DATA_BLOCK "PackMLCfg"   // DB31603
TITLE = CPG_PackMLCfg
{ S7_Optimized_Access := 'TRUE' }
AUTHOR : tech.team.motioncontrol@siemens.com
FAMILY : CPG
VERSION : 1.0
// Support: tech.team.motioncontrol@siemens.com
// Fax: +49 (0) 9131/98-1297
// stored: AutoNumber true, DBAccessibleFromOPCUA true, DBAccessibleFromWebserver true, IsOnlyStoredInLoadMemory false, IsRetainMemResEnabled false, IsWriteProtectedInAS false, MemoryReserve 0
   VAR
      Cfg { S7_SetPoint := 'True'} : "typeLPMLV30_Configuration";   // PackML Configuration Data
      Names { S7_SetPoint := 'True'} : "typeLPMLV30_NamesConfiguration";   // PackML Names Data
      disable : Struct   // Bits used to disable TR88 UN & EMs
         UN : Bool;   // UN (1 = disable, 0= enable)
         EM00 : Struct   // EM00 (1 = disable, 0 = enable)
            EM : Bool;   // EMxx (1 = disable, 0 = enable)
            CM01 : Bool;   // CMxx (1 = disable, 0 = enable)
            CM02 : Bool;   // CMxx (1 = disable, 0 = enable)
            CM03 : Bool;   // CMxx (1 = disable, 0 = enable)
            CM04 : Bool;   // CMxx (1 = disable, 0 = enable)
            CM05 : Bool;   // CMxx (1 = disable, 0 = enable)
            CM06 : Bool;   // CMxx (1 = disable, 0 = enable)
            CM07 : Bool;   // CMxx (1 = disable, 0 = enable)
            CM08 : Bool;   // CMxx (1 = disable, 0 = enable)
            CM09 : Bool;   // CMxx (1 = disable, 0 = enable)
            CM10 : Bool;   // CMxx (1 = disable, 0 = enable)
         END_STRUCT;
         EM01 : Struct   // EM01 (1 = disable, 0 = enable)
            EM : Bool;   // EMxx (1 = disable, 0 = enable)
            CM01 : Bool;   // CMxx (1 = disable, 0 = enable)
            CM02 : Bool;   // CMxx (1 = disable, 0 = enable)
            CM03 : Bool;   // CMxx (1 = disable, 0 = enable)
            CM04 : Bool;   // CMxx (1 = disable, 0 = enable)
            CM05 : Bool;   // CMxx (1 = disable, 0 = enable)
            CM06 : Bool;   // CMxx (1 = disable, 0 = enable)
            CM07 : Bool;   // CMxx (1 = disable, 0 = enable)
            CM08 : Bool;   // CMxx (1 = disable, 0 = enable)
            CM09 : Bool;   // CMxx (1 = disable, 0 = enable)
            CM10 : Bool;   // CMxx (1 = disable, 0 = enable)
         END_STRUCT;
         EM02 : Struct   // EM02 (1 = disable, 0 = enable)
            EM : Bool;   // EMxx (1 = disable, 0 = enable)
            CM01 : Bool;   // CMxx (1 = disable, 0 = enable)
            CM02 : Bool;   // CMxx (1 = disable, 0 = enable)
            CM03 : Bool;   // CMxx (1 = disable, 0 = enable)
            CM04 : Bool;   // CMxx (1 = disable, 0 = enable)
            CM05 : Bool;   // CMxx (1 = disable, 0 = enable)
            CM06 : Bool;   // CMxx (1 = disable, 0 = enable)
            CM07 : Bool;   // CMxx (1 = disable, 0 = enable)
            CM08 : Bool;   // CMxx (1 = disable, 0 = enable)
            CM09 : Bool;   // CMxx (1 = disable, 0 = enable)
            CM10 : Bool;   // CMxx (1 = disable, 0 = enable)
         END_STRUCT;
         EM03 : Struct   // EM03 (1 = disable, 0 = enable)
            EM : Bool;   // EMxx (1 = disable, 0 = enable)
            CM01 : Bool;   // CMxx (1 = disable, 0 = enable)
            CM02 : Bool;   // CMxx (1 = disable, 0 = enable)
            CM03 : Bool;   // CMxx (1 = disable, 0 = enable)
            CM04 : Bool;   // CMxx (1 = disable, 0 = enable)
            CM05 : Bool;   // CMxx (1 = disable, 0 = enable)
            CM06 : Bool;   // CMxx (1 = disable, 0 = enable)
            CM07 : Bool;   // CMxx (1 = disable, 0 = enable)
            CM08 : Bool;   // CMxx (1 = disable, 0 = enable)
            CM09 : Bool;   // CMxx (1 = disable, 0 = enable)
            CM10 : Bool;   // CMxx (1 = disable, 0 = enable)
         END_STRUCT;
         EM04 : Struct   // EM04 (1 = disable, 0 = enable)
            EM : Bool;   // EMxx (1 = disable, 0 = enable)
            CM01 : Bool;   // CMxx (1 = disable, 0 = enable)
            CM02 : Bool;   // CMxx (1 = disable, 0 = enable)
            CM03 : Bool;   // CMxx (1 = disable, 0 = enable)
            CM04 : Bool;   // CMxx (1 = disable, 0 = enable)
            CM05 : Bool;   // CMxx (1 = disable, 0 = enable)
            CM06 : Bool;   // CMxx (1 = disable, 0 = enable)
            CM07 : Bool;   // CMxx (1 = disable, 0 = enable)
            CM08 : Bool;   // CMxx (1 = disable, 0 = enable)
            CM09 : Bool;   // CMxx (1 = disable, 0 = enable)
            CM10 : Bool;   // CMxx (1 = disable, 0 = enable)
         END_STRUCT;
         EM05 : Struct   // EM05 (1 = disable, 0 = enable)
            EM : Bool;   // EMxx (1 = disable, 0 = enable)
            CM01 : Bool;   // CMxx (1 = disable, 0 = enable)
            CM02 : Bool;   // CMxx (1 = disable, 0 = enable)
            CM03 : Bool;   // CMxx (1 = disable, 0 = enable)
            CM04 : Bool;   // CMxx (1 = disable, 0 = enable)
            CM05 : Bool;   // CMxx (1 = disable, 0 = enable)
            CM06 : Bool;   // CMxx (1 = disable, 0 = enable)
            CM07 : Bool;   // CMxx (1 = disable, 0 = enable)
            CM08 : Bool;   // CMxx (1 = disable, 0 = enable)
            CM09 : Bool;   // CMxx (1 = disable, 0 = enable)
            CM10 : Bool;   // CMxx (1 = disable, 0 = enable)
         END_STRUCT;
         EM06 : Struct   // EM06 (1 = disable, 0 = enable)
            EM : Bool;   // EMxx (1 = disable, 0 = enable)
            CM01 : Bool;   // CMxx (1 = disable, 0 = enable)
            CM02 : Bool;   // CMxx (1 = disable, 0 = enable)
            CM03 : Bool;   // CMxx (1 = disable, 0 = enable)
            CM04 : Bool;   // CMxx (1 = disable, 0 = enable)
            CM05 : Bool;   // CMxx (1 = disable, 0 = enable)
            CM06 : Bool;   // CMxx (1 = disable, 0 = enable)
            CM07 : Bool;   // CMxx (1 = disable, 0 = enable)
            CM08 : Bool;   // CMxx (1 = disable, 0 = enable)
            CM09 : Bool;   // CMxx (1 = disable, 0 = enable)
            CM10 : Bool;   // CMxx (1 = disable, 0 = enable)
         END_STRUCT;
         EM07 : Struct   // EM07 (1 = disable, 0 = enable)
            EM : Bool;   // EMxx (1 = disable, 0 = enable)
            CM01 : Bool;   // CMxx (1 = disable, 0 = enable)
            CM02 : Bool;   // CMxx (1 = disable, 0 = enable)
            CM03 : Bool;   // CMxx (1 = disable, 0 = enable)
            CM04 : Bool;   // CMxx (1 = disable, 0 = enable)
            CM05 : Bool;   // CMxx (1 = disable, 0 = enable)
            CM06 : Bool;   // CMxx (1 = disable, 0 = enable)
            CM07 : Bool;   // CMxx (1 = disable, 0 = enable)
            CM08 : Bool;   // CMxx (1 = disable, 0 = enable)
            CM09 : Bool;   // CMxx (1 = disable, 0 = enable)
            CM10 : Bool;   // CMxx (1 = disable, 0 = enable)
         END_STRUCT;
         EM08 : Struct   // EM08 (1 = disable, 0 = enable)
            EM : Bool;   // EMxx (1 = disable, 0 = enable)
            CM01 : Bool;   // CMxx (1 = disable, 0 = enable)
            CM02 : Bool;   // CMxx (1 = disable, 0 = enable)
            CM03 : Bool;   // CMxx (1 = disable, 0 = enable)
            CM04 : Bool;   // CMxx (1 = disable, 0 = enable)
            CM05 : Bool;   // CMxx (1 = disable, 0 = enable)
            CM06 : Bool;   // CMxx (1 = disable, 0 = enable)
            CM07 : Bool;   // CMxx (1 = disable, 0 = enable)
            CM08 : Bool;   // CMxx (1 = disable, 0 = enable)
            CM09 : Bool;   // CMxx (1 = disable, 0 = enable)
            CM10 : Bool;   // CMxx (1 = disable, 0 = enable)
         END_STRUCT;
         EM09 : Struct   // EM09 (1 = disable, 0 = enable)
            EM : Bool;   // EMxx (1 = disable, 0 = enable)
            CM01 : Bool;   // CMxx (1 = disable, 0 = enable)
            CM02 : Bool;   // CMxx (1 = disable, 0 = enable)
            CM03 : Bool;   // CMxx (1 = disable, 0 = enable)
            CM04 : Bool;   // CMxx (1 = disable, 0 = enable)
            CM05 : Bool;   // CMxx (1 = disable, 0 = enable)
            CM06 : Bool;   // CMxx (1 = disable, 0 = enable)
            CM07 : Bool;   // CMxx (1 = disable, 0 = enable)
            CM08 : Bool;   // CMxx (1 = disable, 0 = enable)
            CM09 : Bool;   // CMxx (1 = disable, 0 = enable)
            CM10 : Bool;   // CMxx (1 = disable, 0 = enable)
         END_STRUCT;
      END_STRUCT;
   END_VAR
BEGIN
   Names.unitModesNames[2,0] := 'Invalid';
   Names.unitModesNames[2,1] := 'Production';
   Names.unitModesNames[2,2] := 'Maintenance';
   Names.unitModesNames[2,3] := 'Manual';
   Names.unitModesNames[2,4] := 'User Mode 01';
   Names.statesNames[1,1] := 'Clearing';
   Names.statesNames[1,2] := 'Stopped';
   Names.statesNames[1,3] := 'Starting';
   Names.statesNames[1,4] := 'Idle';
   Names.statesNames[1,5] := 'Suspended';
   Names.statesNames[1,6] := 'Execute';
   Names.statesNames[1,7] := 'Stopping';
   Names.statesNames[1,8] := 'Aborting';
   Names.statesNames[1,9] := 'Aborted';
   Names.statesNames[1,10] := 'Holding';
   Names.statesNames[1,11] := 'Held';
   Names.statesNames[1,12] := 'UnHolding';
   Names.statesNames[1,13] := 'Suspending';
   Names.statesNames[1,14] := 'UnSuspending';
   Names.statesNames[1,15] := 'Resetting';
   Names.statesNames[1,16] := 'Completing';
   Names.statesNames[1,17] := 'Complete';
   Names.statesNames[2,0] := 'Undefined';
   Names.statesNames[2,1] := 'Limpiar';
   Names.statesNames[2,2] := 'Detenido';
   Names.statesNames[2,3] := 'Empezando';
   Names.statesNames[2,4] := 'Parado';
   Names.statesNames[2,5] := 'Interrumpido';
   Names.statesNames[2,6] := 'Correr';
   Names.statesNames[2,7] := 'Detener';
   Names.statesNames[2,8] := 'Anulando';
   Names.statesNames[2,9] := 'Anulado';
   Names.statesNames[2,10] := 'Mantener';
   Names.statesNames[2,11] := 'Mantenido';
   Names.statesNames[2,12] := 'Desmentener';
   Names.statesNames[2,13] := 'Interrumpir';
   Names.statesNames[2,14] := 'Desinterrumpir';
   Names.statesNames[2,15] := 'Reajustar';
   Names.statesNames[2,16] := 'Terminar';
   Names.statesNames[2,17] := 'Terminado';
END_DATA_BLOCK

DATA_BLOCK "RecipeCfg"   // DB1605
TITLE = CPG_RecipeCfg
{ S7_Optimized_Access := 'TRUE' }
AUTHOR : tech.team.motioncontrol@siemens.com
FAMILY : CPG
VERSION : 1.1
// Support: tech.team.motioncontrol@siemens.com
// stored: AutoNumber true, DBAccessibleFromOPCUA true, DBAccessibleFromWebserver true, IsOnlyStoredInLoadMemory false, IsRetainMemResEnabled false, IsWriteProtectedInAS false, MemoryReserve 0
   VAR
      setpoints_REAL { S7_SetPoint := 'True'} : Array[0.."CPG_NO_OF_SETPOINT_REAL_UPPER_LIM"] of "CPG_typeRecipeSetpoint_REAL";   // Array of setpoints of REAL
      setpoints_DINT { S7_SetPoint := 'True'} : Array[0.."CPG_NO_OF_SETPOINT_DINT_UPPER_LIM"] of "CPG_typeRecipeSetpoint_DINT";   // Array of setpoints of DINT
      setpoints_BOOL { S7_SetPoint := 'True'} : Array[0.."CPG_NO_OF_SETPOINT_BOOL_UPPER_LIM"] of "CPG_typeRecipeSetpoint_BOOL";   // Array of setpoints of BOOL
      setpoints_STRING { S7_SetPoint := 'True'} : Array[0.."CPG_NO_OF_SETPOINT_STRING_UPPER_LIM"] of "CPG_typeRecipeSetpoint_STRING";   // Array of setpoints of STRING
      recipeControl { S7_SetPoint := 'True'} : "CPG_typeRecipeControl";   // FB_Recipe_Control communicates to the setpoints via this tag
      recipeNames : Array[0.."CPG_NO_OF_RECIPE_UPPER_LIM"] of String[60];   // Array holding the names of all recipes
      recipeCumTimes : Array[0.."CPG_NO_OF_RECIPE_UPPER_LIM"] of Time;   // Array holding the cumulative time all recipes have been active
      recipeLastSaveTimes : Array[0.."CPG_NO_OF_RECIPE_UPPER_LIM"] of DTL;   // Array holding the last time each recipe was saved
   END_VAR
BEGIN
   setpoints_REAL[0].SetpointName[0] := 'LH 1 Length';
   setpoints_DINT[0].SetpointName[0] := 'DINT SP 0';
   setpoints_BOOL[0].SetpointName[0] := 'BOOL SP 0';
   setpoints_BOOL[0].SetpointName[1] := '';
   setpoints_BOOL[0].Text_True[0] := 'TRUE';
   setpoints_BOOL[0].Text_True[1] := '';
   setpoints_BOOL[0].Text_False[0] := 'FALSE';
   setpoints_STRING[0].RecipeValues[0] := 'a';
   setpoints_STRING[0].RecipeValues[1] := 'b';
   setpoints_STRING[0].RecipeValues[2] := 'c';
   setpoints_STRING[0].RecipeValues[3] := 'd';
   setpoints_STRING[0].RecipeValues[4] := 'e';
   setpoints_STRING[0].RecipeValues[5] := 'f';
   setpoints_STRING[0].RecipeValues[6] := 'g';
   setpoints_STRING[0].SetpointName[0] := 'STRING SP 0';
   recipeControl.CurrentRecipeID := 0;
   recipeControl.CurrentRecipeName := 'Recipe 0';
   recipeControl.RecipeID_A := 1;
   recipeControl.RecipeID_B := 2;
   recipeControl.RecipeID_C := 3;
   recipeNames[0] := 'Recipe 0';
   recipeNames[1] := 'Recipe 1';
   recipeNames[2] := 'Recipe 2';
   recipeNames[3] := 'Recipe 3';
   recipeNames[4] := 'Recipe 4';
   recipeNames[5] := 'Recipe 5';
   recipeNames[6] := 'Recipe 6';
   recipeNames[7] := 'Recipe 7';
   recipeNames[8] := 'Recipe 8';
   recipeNames[9] := 'Recipe 9';
   recipeNames[10] := 'Recipe 10';
   recipeNames[11] := 'Recipe 11';
   recipeNames[12] := 'Recipe 12';
   recipeNames[13] := 'Recipe 13';
   recipeNames[14] := 'Recipe 14';
   recipeNames[15] := 'Recipe 15';
   recipeNames[16] := 'Recipe 16';
   recipeNames[17] := 'Recipe 17';
   recipeNames[18] := 'Recipe 18';
   recipeNames[19] := 'Recipe 19';
   recipeNames[20] := 'Recipe 20';
   recipeLastSaveTimes[0..20] := DTL#2019-1-1-00:00:00;
END_DATA_BLOCK

DATA_BLOCK "StatusCfg"   // DB31602
TITLE = CPG_StatusCfg
{ S7_Optimized_Access := 'TRUE' }
AUTHOR : tech.team.motioncontrol@siemens.com
FAMILY : CPG
VERSION : 1.0
// Support: tech.team.motioncontrol@siemens.com
// Fax: +49 (0) 9131/98-1297
// stored: AutoNumber true, DBAccessibleFromOPCUA true, DBAccessibleFromWebserver true, IsOnlyStoredInLoadMemory false, IsRetainMemResEnabled false, IsWriteProtectedInAS false, MemoryReserve 0
   VAR
      Event { ExternalAccessible := 'False'; ExternalVisible := 'False'; ExternalWritable := 'False'; S7_SetPoint := 'True'} : Array[0.."CPG_NO_OF_CFG_STATUS_UPPER_LIM"] of "CPG_typeEventCfg";
   END_VAR
BEGIN
   // Event[0] : Status Test
   // Event[1] : 'Alarms Present'
   // Event[2] : 'Waiting for Reset Cmd'
   // Event[3] : 'Waiting for Start Cmd'
   // Event[4] : 'Not Ready for Motion'
   // Event[5] : 'Waiting for No Motion'
   // Event[6] : 'Waiting to start Gearing'
   // Event[7] : 'Waiting to Finish'
   // Event[8] : 'Waiting for Un-Hold Cmd'
   // Event[9] : 'Waiting for Mat. Supply'
   // Event[10] : Spare
   // Event[11] : Spare
   // Event[12] : Spare
   // Event[13] : Spare
   // Event[14] : Spare
   // Event[15] : Spare
   // Event[16] : Spare
   // Event[17] : Spare
   // Event[18] : Spare
   // Event[19] : Spare
   Event[0].ID := 0;
   Event[1].ID := 1;
   Event[2].ID := 2;
   Event[3].ID := 3;
   Event[4].ID := 4;
   Event[5].ID := 5;
   Event[6].ID := 6;
   Event[7].ID := 7;
   Event[8].ID := 8;
   Event[9].ID := 9;
   Event[10].ID := 10;
   Event[11].ID := 11;
   Event[12].ID := 12;
   Event[13].ID := 13;
   Event[14].ID := 14;
   Event[15].ID := 15;
   Event[16].ID := 16;
   Event[17].ID := 17;
   Event[18].ID := 18;
   Event[19].ID := 19;
   Event[0].message[0..1] := 'Status Test';
   Event[0].message[2] := 'Los Status Test';
   Event[1].message[0] := 'Alarms Present';
   Event[1].message[1] := 'Alarme anstehend';
   Event[1].message[2] := 'Las Alarms Present';
   Event[2].message[0] := 'Waiting for Reset PB';
   Event[2].message[1] := 'Warte auf Reset Taste';
   Event[2].message[2] := 'Esperando de Reajustar PB';
   Event[3].message[0] := 'Waiting for Start PB';
   Event[3].message[1] := 'Warten auf Start Taste';
   Event[3].message[2] := 'Esperando de Comenzar PB';
   Event[4].message[0] := 'Not Ready for Motion';
   Event[4].message[1] := 'Maschine nicht anlaufbereit';
   Event[4].message[2] := 'No Listo para Movimiento';
   Event[5].message[0] := 'Waiting for No Motion';
   Event[5].message[1] := 'Warte auf Maschinenstillstand';
   Event[5].message[2] := 'Esperando No Movimiento';
   Event[6].message[0] := 'Waiting to start Gearing';
   Event[6].message[1] := 'Warte auf Start Getriebegleichlauf';
   Event[6].message[2] := 'Waiting to start Gearing';
   Event[7].message[0] := 'Waiting to Finish';
   Event[7].message[1] := 'Warte auf Ende Leerfahren';
   Event[7].message[2] := 'Esperando para Terminar';
   Event[8].message[0] := 'Waiting for Un-Hold PB';
   Event[8].message[1] := 'Warte auf Un-Hold Taste';
   Event[8].message[2] := 'Waiting for Un-Hold PB';
   Event[9].message[0] := 'Waiting for Mat. Supply';
   Event[9].message[1] := 'Warte auf Materialversorgung';
   Event[9].message[2] := 'Waiting for Mat. Supply';
   Event[10].message[0] := 'Spare';
   Event[10].message[1] := 'Reserve';
   Event[10].message[2] := 'Spare';
   Event[11].message[0] := 'Spare';
   Event[11].message[1] := 'Reserve';
   Event[11].message[2] := 'Spare';
   Event[12].message[0] := 'Spare';
   Event[12].message[1] := 'Reserve';
   Event[12].message[2] := 'Spare';
   Event[13].message[0] := 'Spare';
   Event[13].message[1] := 'Reserve';
   Event[13].message[2] := 'Spare';
   Event[14].message[0] := 'Spare';
   Event[14].message[1] := 'Reserve';
   Event[14].message[2] := 'Spare';
   Event[15].message[0] := 'Spare';
   Event[15].message[1] := 'Reserve';
   Event[15].message[2] := 'Spare';
   Event[16].message[0] := 'Spare';
   Event[16].message[1] := 'Reserve';
   Event[16].message[2] := 'Spare';
   Event[17].message[0] := 'Spare';
   Event[17].message[1] := 'Reserve';
   Event[17].message[2] := 'Spare';
   Event[18].message[0] := 'Spare';
   Event[18].message[1] := 'Reserve';
   Event[18].message[2] := 'Spare';
   Event[19].message[0] := 'Spare';
   Event[19].message[1] := 'Reserve';
   Event[19].message[2] := 'Spare';
END_DATA_BLOCK

DATA_BLOCK "WarningCfg"   // DB31601
TITLE = CPG_WarningCfg
{ S7_Optimized_Access := 'TRUE' }
AUTHOR : tech.team.motioncontrol@siemens.com
FAMILY : CPG
VERSION : 1.0
// Support: tech.team.motioncontrol@siemens.com
// Fax: +49 (0) 9131/98-1297
// stored: AutoNumber true, DBAccessibleFromOPCUA true, DBAccessibleFromWebserver true, IsOnlyStoredInLoadMemory false, IsRetainMemResEnabled false, IsWriteProtectedInAS false, MemoryReserve 0
   VAR
      Event { ExternalAccessible := 'False'; ExternalVisible := 'False'; ExternalWritable := 'False'; S7_SetPoint := 'True'} : Array[0.."CPG_NO_OF_CFG_WARNINGS_UPPER_LIM"] of "CPG_typeEventCfg";
   END_VAR
BEGIN
   // Event[0] : Warning Test
   // Event[1] : Low Bottle Supply
   // Event[2] : Low Label Supply
   // Event[3] : Spare
   // Event[4] : Spare
   // Event[5] : Spare
   // Event[6] : Spare
   // Event[7] : Spare
   // Event[8] : Spare
   // Event[9] : Spare
   // Event[10] : Spare
   // Event[11] : Spare
   // Event[12] : Spare
   // Event[13] : Spare
   // Event[14] : Spare
   // Event[15] : Spare
   // Event[16] : Spare
   // Event[17] : Spare
   // Event[18] : Spare
   // Event[19] : Spare
   // Event[20] : Spare
   // Event[21] : Spare
   // Event[22] : Spare
   // Event[23] : Spare
   // Event[24] : Spare
   // Event[25] : Spare
   // Event[26] : Spare
   // Event[27] : Spare
   // Event[28] : Spare
   // Event[29] : Spare
   Event[0].ID := 0;
   Event[1].ID := 1;
   Event[2].ID := 2;
   Event[3].ID := 3;
   Event[4].ID := 4;
   Event[5].ID := 5;
   Event[6].ID := 6;
   Event[7].ID := 7;
   Event[8].ID := 8;
   Event[9].ID := 9;
   Event[10].ID := 10;
   Event[11].ID := 11;
   Event[12].ID := 12;
   Event[13].ID := 13;
   Event[14].ID := 14;
   Event[15].ID := 15;
   Event[16].ID := 16;
   Event[17].ID := 17;
   Event[18].ID := 18;
   Event[19].ID := 19;
   Event[20].ID := 20;
   Event[21].ID := 21;
   Event[22].ID := 22;
   Event[23].ID := 23;
   Event[24].ID := 24;
   Event[25].ID := 25;
   Event[26].ID := 26;
   Event[27].ID := 27;
   Event[28].ID := 28;
   Event[29].ID := 29;
   Event[0].message[0..1] := 'Warning Test';
   Event[0].message[2] := 'Los Warning Test';
   Event[1].message[0] := 'Low Bottle Supply';
   Event[1].message[1] := 'Flaschenzufuhr niedrig';
   Event[1].message[2] := 'Las Low Bottle Supply';
   Event[2].message[0] := 'Low Label Supply';
   Event[2].message[1] := 'Etikettenzufuhr niedrig';
   Event[2].message[2] := 'Las Low Label Supply';
   Event[3].message[0] := 'Spare';
   Event[3].message[1] := 'Reserve';
   Event[3].message[2] := 'Spare';
   Event[4].message[0] := 'Spare';
   Event[4].message[1] := 'Reserve';
   Event[4].message[2] := 'Spare';
   Event[5].message[0] := 'Spare';
   Event[5].message[1] := 'Reserve';
   Event[5].message[2] := 'Spare';
   Event[6].message[0] := 'Spare';
   Event[6].message[1] := 'Reserve';
   Event[6].message[2] := 'Spare';
   Event[7].message[0] := 'Spare';
   Event[7].message[1] := 'Reserve';
   Event[7].message[2] := 'Spare';
   Event[8].message[0] := 'Spare';
   Event[8].message[1] := 'Reserve';
   Event[8].message[2] := 'Spare';
   Event[9].message[0] := 'Spare';
   Event[9].message[1] := 'Reserve';
   Event[9].message[2] := 'Spare';
   Event[10].message[0] := 'Spare';
   Event[10].message[1] := 'Reserve';
   Event[10].message[2] := 'Spare';
   Event[11].message[0] := 'Spare';
   Event[11].message[1] := 'Reserve';
   Event[11].message[2] := 'Spare';
   Event[12].message[0] := 'Spare';
   Event[12].message[1] := 'Reserve';
   Event[12].message[2] := 'Spare';
   Event[13].message[0] := 'Spare';
   Event[13].message[1] := 'Reserve';
   Event[13].message[2] := 'Spare';
   Event[14].message[0] := 'Spare';
   Event[14].message[1] := 'Reserve';
   Event[14].message[2] := 'Spare';
   Event[15].message[0] := 'Spare';
   Event[15].message[1] := 'Reserve';
   Event[15].message[2] := 'Spare';
   Event[16].message[0] := 'Spare';
   Event[16].message[1] := 'Reserve';
   Event[16].message[2] := 'Spare';
   Event[17].message[0] := 'Spare';
   Event[17].message[1] := 'Reserve';
   Event[17].message[2] := 'Spare';
   Event[18].message[0] := 'Spare';
   Event[18].message[1] := 'Reserve';
   Event[18].message[2] := 'Spare';
   Event[19].message[0] := 'Spare';
   Event[19].message[1] := 'Reserve';
   Event[19].message[2] := 'Spare';
   Event[20].message[0] := 'Spare';
   Event[20].message[1] := 'Reserve';
   Event[20].message[2] := 'Spare';
   Event[21].message[0] := 'Spare';
   Event[21].message[1] := 'Reserve';
   Event[21].message[2] := 'Spare';
   Event[22].message[0] := 'Spare';
   Event[22].message[1] := 'Reserve';
   Event[22].message[2] := 'Spare';
   Event[23].message[0] := 'Spare';
   Event[23].message[1] := 'Reserve';
   Event[23].message[2] := 'Spare';
   Event[24].message[0] := 'Spare';
   Event[24].message[1] := 'Reserve';
   Event[24].message[2] := 'Spare';
   Event[25].message[0] := 'Spare';
   Event[25].message[1] := 'Reserve';
   Event[25].message[2] := 'Spare';
   Event[26].message[0] := 'Spare';
   Event[26].message[1] := 'Reserve';
   Event[26].message[2] := 'Spare';
   Event[27].message[0] := 'Spare';
   Event[27].message[1] := 'Reserve';
   Event[27].message[2] := 'Spare';
   Event[28].message[0] := 'Spare';
   Event[28].message[1] := 'Reserve';
   Event[28].message[2] := 'Spare';
   Event[29].message[0] := 'Spare';
   Event[29].message[1] := 'Reserve';
   Event[29].message[2] := 'Spare';
END_DATA_BLOCK

ORGANIZATION_BLOCK "Main"   // OB1, LAD, ProgramCycle
TITLE = Main
{ S7_Optimized_Access := 'TRUE' }
AUTHOR : tech.team.motioncontrol@siemens.com
FAMILY : CPG
VERSION : 1.0
// Support: tech.team.motioncontrol@siemens.com
// Fax: +49 (0) 9131/98-1297
// stored: AutoNumber true, IsIECCheckEnabled false, SetENOAutomatically false
   VAR_INPUT
      Initial_Call : Bool;   // Initial call of this OB
      Remanence : Bool;   // =True, if remanent data are available
   END_VAR
   VAR_TEMP   // added for the SCL form of the ladder/FBD networks
      _w1 : Bool;
   END_VAR
BEGIN

REGION Network 1: Factory IO PLCSIM Communication
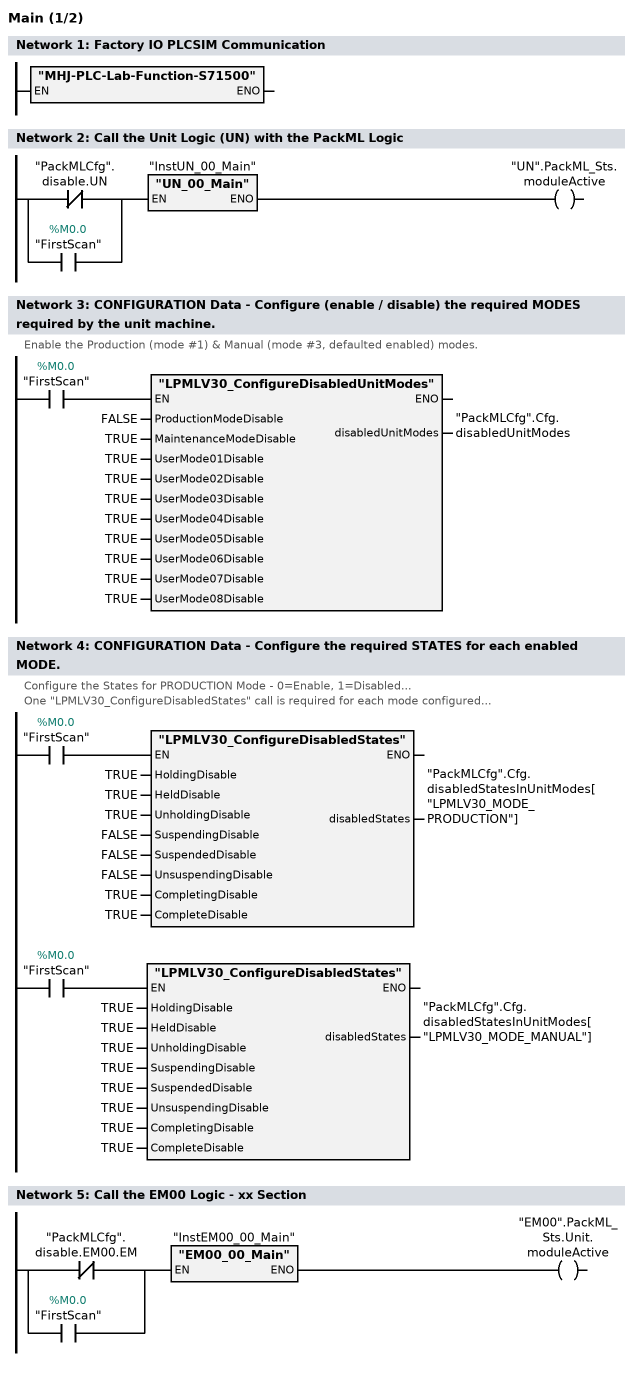
   RUNG wire#powerrail
      "MHJ-PLC-Lab-Function-S71500"()
   END_RUNG
   // the same network as SCL:
   "MHJ-PLC-Lab-Function-S71500"();
END_REGION

REGION Network 2: Call the Unit Logic (UN) with the PackML Logic
   RUNG wire#powerrail
      I_Contact( "PackMLCfg".disable.UN )
      wire#w1
      "InstUN_00_Main"()
      Coil( "UN".PackML_Sts.moduleActive )
   END_RUNG
   RUNG wire#powerrail
      Contact( "FirstScan" )
   END_RUNG wire#w1
   // the same network as SCL:
   "InstUN_00_Main"(EN := NOT "PackMLCfg".disable.UN OR "FirstScan", ENO => #_w1);   // "UN_00_Main"
   "UN".PackML_Sts.moduleActive := #_w1;
END_REGION

REGION Network 3: CONFIGURATION Data - Configure (enable / disable) the required MODES required by the unit machine.
   // Enable the Production (mode #1) & Manual (mode #3, defaulted enabled) modes.
   RUNG wire#powerrail
      Contact( "FirstScan" )
      "LPMLV30_ConfigureDisabledUnitModes"(ProductionModeDisable := FALSE, MaintenanceModeDisable := TRUE, UserMode01Disable := TRUE, UserMode02Disable := TRUE, UserMode03Disable := TRUE, UserMode04Disable := TRUE, UserMode05Disable := TRUE, UserMode06Disable := TRUE, UserMode07Disable := TRUE, UserMode08Disable := TRUE, disabledUnitModes => "PackMLCfg".Cfg.disabledUnitModes)
   END_RUNG
   // the same network as SCL:
   IF "FirstScan" THEN
       "LPMLV30_ConfigureDisabledUnitModes"(ProductionModeDisable := FALSE,
                               MaintenanceModeDisable := TRUE,
                               UserMode01Disable := TRUE,
                               UserMode02Disable := TRUE,
                               UserMode03Disable := TRUE,
                               UserMode04Disable := TRUE,
                               UserMode05Disable := TRUE,
                               UserMode06Disable := TRUE,
                               UserMode07Disable := TRUE,
                               UserMode08Disable := TRUE,
                               disabledUnitModes => "PackMLCfg".Cfg.disabledUnitModes);
   END_IF;
END_REGION

REGION Network 4: CONFIGURATION Data - Configure the required STATES for each enabled MODE.
   // Configure the States for PRODUCTION Mode - 0=Enable, 1=Disabled...
   // One "LPMLV30_ConfigureDisabledStates" call is required for each mode configured...
   RUNG wire#powerrail
      Contact( "FirstScan" )
      "LPMLV30_ConfigureDisabledStates"(HoldingDisable := TRUE, HeldDisable := TRUE, UnholdingDisable := TRUE, SuspendingDisable := FALSE, SuspendedDisable := FALSE, UnsuspendingDisable := FALSE, CompletingDisable := TRUE, CompleteDisable := TRUE, disabledStates => "PackMLCfg".Cfg.disabledStatesInUnitModes["LPMLV30_MODE_PRODUCTION"])
   END_RUNG
   RUNG wire#powerrail
      Contact( "FirstScan" )
      "LPMLV30_ConfigureDisabledStates"(HoldingDisable := TRUE, HeldDisable := TRUE, UnholdingDisable := TRUE, SuspendingDisable := TRUE, SuspendedDisable := TRUE, UnsuspendingDisable := TRUE, CompletingDisable := TRUE, CompleteDisable := TRUE, disabledStates => "PackMLCfg".Cfg.disabledStatesInUnitModes["LPMLV30_MODE_MANUAL"])
   END_RUNG
   // the same network as SCL:
   IF "FirstScan" THEN
       "LPMLV30_ConfigureDisabledStates"(HoldingDisable := TRUE,
                               HeldDisable := TRUE,
                               UnholdingDisable := TRUE,
                               SuspendingDisable := FALSE,
                               SuspendedDisable := FALSE,
                               UnsuspendingDisable := FALSE,
                               CompletingDisable := TRUE,
                               CompleteDisable := TRUE,
                               disabledStates => "PackMLCfg".Cfg.disabledStatesInUnitModes["LPMLV30_MODE_PRODUCTION"]);
   END_IF;
   IF "FirstScan" THEN
       "LPMLV30_ConfigureDisabledStates"(HoldingDisable := TRUE,
                               HeldDisable := TRUE,
                               UnholdingDisable := TRUE,
                               SuspendingDisable := TRUE,
                               SuspendedDisable := TRUE,
                               UnsuspendingDisable := TRUE,
                               CompletingDisable := TRUE,
                               CompleteDisable := TRUE,
                               disabledStates => "PackMLCfg".Cfg.disabledStatesInUnitModes["LPMLV30_MODE_MANUAL"]);
   END_IF;
END_REGION

REGION Network 5: Call the EM00 Logic - xx Section
   RUNG wire#powerrail
      I_Contact( "PackMLCfg".disable.EM00.EM )
      wire#w1
      "InstEM00_00_Main"()
      Coil( "EM00".PackML_Sts.Unit.moduleActive )
   END_RUNG
   RUNG wire#powerrail
      Contact( "FirstScan" )
   END_RUNG wire#w1
   // the same network as SCL:
   "InstEM00_00_Main"(EN := NOT "PackMLCfg".disable.EM00.EM OR "FirstScan", ENO => #_w1);   // "EM00_00_Main"
   "EM00".PackML_Sts.Unit.moduleActive := #_w1;
END_REGION

REGION Network 6: Call the EM01 Logic - xx Section
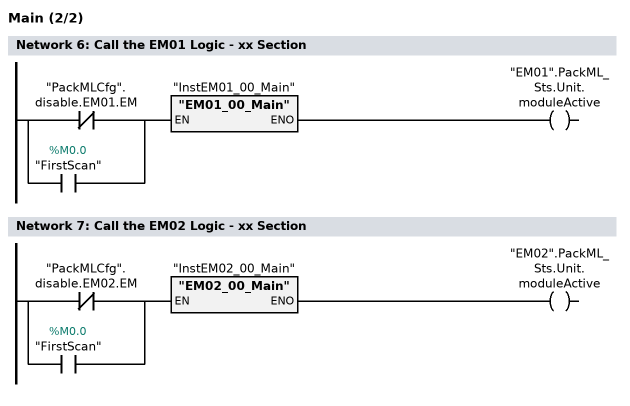
   RUNG wire#powerrail
      I_Contact( "PackMLCfg".disable.EM01.EM )
      wire#w1
      "InstEM01_00_Main"()
      Coil( "EM01".PackML_Sts.Unit.moduleActive )
   END_RUNG
   RUNG wire#powerrail
      Contact( "FirstScan" )
   END_RUNG wire#w1
   // the same network as SCL:
   "InstEM01_00_Main"(EN := NOT "PackMLCfg".disable.EM01.EM OR "FirstScan", ENO => #_w1);   // "EM01_00_Main"
   "EM01".PackML_Sts.Unit.moduleActive := #_w1;
END_REGION

REGION Network 7: Call the EM02 Logic - xx Section
   RUNG wire#powerrail
      I_Contact( "PackMLCfg".disable.EM02.EM )
      wire#w1
      "InstEM02_00_Main"()
      Coil( "EM02".PackML_Sts.Unit.moduleActive )
   END_RUNG
   RUNG wire#powerrail
      Contact( "FirstScan" )
   END_RUNG wire#w1
   // the same network as SCL:
   "InstEM02_00_Main"(EN := NOT "PackMLCfg".disable.EM02.EM OR "FirstScan", ENO => #_w1);   // "EM02_00_Main"
   "EM02".PackML_Sts.Unit.moduleActive := #_w1;
END_REGION
END_ORGANIZATION_BLOCK

FUNCTION_BLOCK "UN_00_Main"   // FB31620, LAD
TITLE = UN_00_Main
{ S7_Optimized_Access := 'TRUE' }
AUTHOR : tech.team.motioncontrol@siemens.com
FAMILY : CPG
VERSION : 1.0
// Support: tech.team.motioncontrol@siemens.com
// Fax: +49 (0) 9131/98-1297
// stored: AutoNumber true, IsIECCheckEnabled false, IsRetainMemResEnabled false, MemoryReserve 100, SetENOAutomatically false, UDAEnableTagReadback false
   VAR
      instPackML_ModuleSum { ExternalAccessible := 'False'; ExternalVisible := 'False'; ExternalWritable := 'False'; S7_SetPoint := 'True'} : "UN_01_PackML_ModuleSum";   // PackML Module Summation Logic of EM-level command and state complete's to unit level
      instPackML { ExternalAccessible := 'False'; ExternalVisible := 'False'; ExternalWritable := 'False'; S7_SetPoint := 'True'} : "UN_02_PackML";
      instLineComm { ExternalAccessible := 'False'; ExternalVisible := 'False'; ExternalWritable := 'False'; S7_SetPoint := 'True'} : "UN_03_LineComm";
      instEventControl { ExternalAccessible := 'False'; ExternalVisible := 'False'; ExternalWritable := 'False'; S7_SetPoint := 'True'} : "UN_04_EventControl";
      instEventSummation { ExternalAccessible := 'False'; ExternalVisible := 'False'; ExternalWritable := 'False'; S7_SetPoint := 'True'} : "UN_05_EventSummation";
      instMiscFunctions { ExternalAccessible := 'False'; ExternalVisible := 'False'; ExternalWritable := 'False'; S7_SetPoint := 'True'} : "UN_06_MiscFunctions";
      instRecipeControl { ExternalAccessible := 'False'; ExternalVisible := 'False'; ExternalWritable := 'False'; S7_SetPoint := 'True'} : "UN_07_RecipeControl";
   END_VAR
   VAR_TEMP   // added for the SCL form of the ladder/FBD networks
      _w1 : Bool;
   END_VAR
BEGIN

REGION Network 1: Call the PackML Module Summation Logic
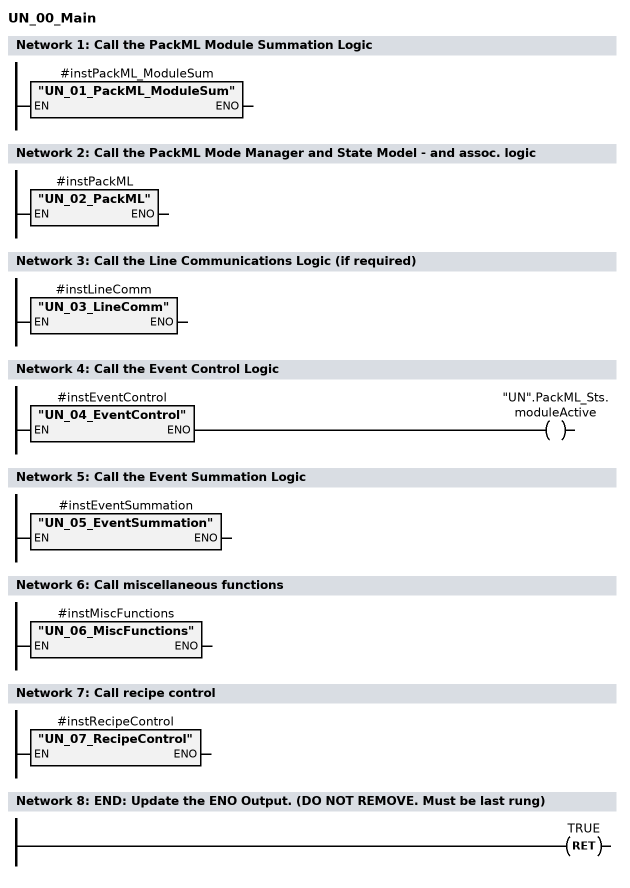
   RUNG wire#powerrail
      #instPackML_ModuleSum()
   END_RUNG
   // the same network as SCL:
   #instPackML_ModuleSum();   // "UN_01_PackML_ModuleSum"
END_REGION

REGION Network 2: Call the PackML Mode Manager and State Model - and assoc. logic
   RUNG wire#powerrail
      #instPackML()
   END_RUNG
   // the same network as SCL:
   #instPackML();   // "UN_02_PackML"
END_REGION

REGION Network 3: Call the Line Communications Logic (if required)
   RUNG wire#powerrail
      #instLineComm()
   END_RUNG
   // the same network as SCL:
   #instLineComm();   // "UN_03_LineComm"
END_REGION

REGION Network 4: Call the Event Control Logic
   RUNG wire#powerrail
      #instEventControl()
      Coil( "UN".PackML_Sts.moduleActive )
   END_RUNG
   // the same network as SCL:
   #instEventControl(ENO => #_w1);   // "UN_04_EventControl"
   "UN".PackML_Sts.moduleActive := #_w1;
END_REGION

REGION Network 5: Call the Event Summation Logic
   RUNG wire#powerrail
      #instEventSummation()
   END_RUNG
   // the same network as SCL:
   #instEventSummation();   // "UN_05_EventSummation"
END_REGION

REGION Network 6: Call miscellaneous functions
   RUNG wire#powerrail
      #instMiscFunctions()
   END_RUNG
   // the same network as SCL:
   #instMiscFunctions();   // "UN_06_MiscFunctions"
END_REGION

REGION Network 7: Call recipe control
   RUNG wire#powerrail
      #instRecipeControl()
   END_RUNG
   // the same network as SCL:
   #instRecipeControl();   // "UN_07_RecipeControl"
END_REGION

REGION Network 8: END: Update the ENO Output. (DO NOT REMOVE. Must be last rung)
   RUNG wire#powerrail
      ReturnCoil( TRUE )
   END_RUNG
   // the same network as SCL:
   ENO := TRUE;
   RETURN;
END_REGION
END_FUNCTION_BLOCK

FUNCTION_BLOCK "UN_01_PackML_ModuleSum"   // FB31621, LAD
TITLE = UN_01_PackML_ModuleSummation
{ S7_Optimized_Access := 'TRUE' }
AUTHOR : tech.team.motioncontrol@siemens.com
FAMILY : CPG
VERSION : 1.0
// Support: tech.team.motioncontrol@siemens.com
// Fax: +49 (0) 9131/98-1297
// stored: AutoNumber true, IsIECCheckEnabled false, IsRetainMemResEnabled false, MemoryReserve 100, SetENOAutomatically false, UDAEnableTagReadback false
   VAR
      statDummyBool { ExternalAccessible := 'False'; ExternalVisible := 'False'; ExternalWritable := 'False'} : Bool;   // dummy bool - placeholder
   END_VAR
BEGIN

REGION Network 1: UN - Reset Command
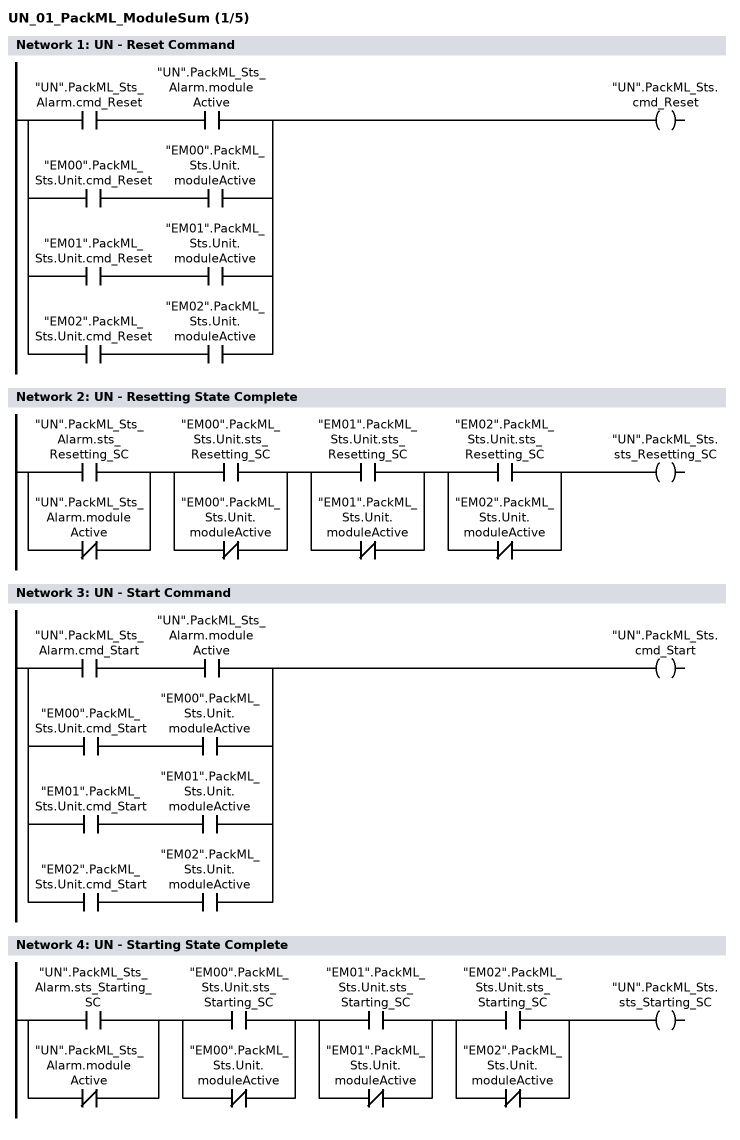
   RUNG wire#powerrail
      Contact( "UN".PackML_Sts_Alarm.cmd_Reset )
      Contact( "UN".PackML_Sts_Alarm.moduleActive )
      wire#w1
      Coil( "UN".PackML_Sts.cmd_Reset )
   END_RUNG
   RUNG wire#powerrail
      Contact( "EM00".PackML_Sts.Unit.cmd_Reset )
      Contact( "EM00".PackML_Sts.Unit.moduleActive )
   END_RUNG wire#w1
   RUNG wire#powerrail
      Contact( "EM01".PackML_Sts.Unit.cmd_Reset )
      Contact( "EM01".PackML_Sts.Unit.moduleActive )
   END_RUNG wire#w1
   RUNG wire#powerrail
      Contact( "EM02".PackML_Sts.Unit.cmd_Reset )
      Contact( "EM02".PackML_Sts.Unit.moduleActive )
   END_RUNG wire#w1
   // the same network as SCL:
   "UN".PackML_Sts.cmd_Reset := ("UN".PackML_Sts_Alarm.cmd_Reset AND "UN".PackML_Sts_Alarm.moduleActive) OR ("EM00".PackML_Sts.Unit.cmd_Reset AND "EM00".PackML_Sts.Unit.moduleActive) OR ("EM01".PackML_Sts.Unit.cmd_Reset AND "EM01".PackML_Sts.Unit.moduleActive) OR ("EM02".PackML_Sts.Unit.cmd_Reset AND "EM02".PackML_Sts.Unit.moduleActive);
END_REGION

REGION Network 2: UN - Resetting State Complete
   RUNG wire#powerrail
      Contact( "UN".PackML_Sts_Alarm.sts_Resetting_SC )
      wire#w1
      Contact( "EM00".PackML_Sts.Unit.sts_Resetting_SC )
      wire#w2
      Contact( "EM01".PackML_Sts.Unit.sts_Resetting_SC )
      wire#w3
      Contact( "EM02".PackML_Sts.Unit.sts_Resetting_SC )
      wire#w4
      Coil( "UN".PackML_Sts.sts_Resetting_SC )
   END_RUNG
   RUNG wire#powerrail
      I_Contact( "UN".PackML_Sts_Alarm.moduleActive )
   END_RUNG wire#w1
   RUNG wire#w1
      I_Contact( "EM00".PackML_Sts.Unit.moduleActive )
   END_RUNG wire#w2
   RUNG wire#w2
      I_Contact( "EM01".PackML_Sts.Unit.moduleActive )
   END_RUNG wire#w3
   RUNG wire#w3
      I_Contact( "EM02".PackML_Sts.Unit.moduleActive )
   END_RUNG wire#w4
   // the same network as SCL:
   "UN".PackML_Sts.sts_Resetting_SC := ("UN".PackML_Sts_Alarm.sts_Resetting_SC OR NOT "UN".PackML_Sts_Alarm.moduleActive) AND ("EM00".PackML_Sts.Unit.sts_Resetting_SC OR NOT "EM00".PackML_Sts.Unit.moduleActive) AND ("EM01".PackML_Sts.Unit.sts_Resetting_SC OR NOT "EM01".PackML_Sts.Unit.moduleActive) AND ("EM02".PackML_Sts.Unit.sts_Resetting_SC OR NOT "EM02".PackML_Sts.Unit.moduleActive);
END_REGION

REGION Network 3: UN - Start Command
   RUNG wire#powerrail
      Contact( "UN".PackML_Sts_Alarm.cmd_Start )
      Contact( "UN".PackML_Sts_Alarm.moduleActive )
      wire#w1
      Coil( "UN".PackML_Sts.cmd_Start )
   END_RUNG
   RUNG wire#powerrail
      Contact( "EM00".PackML_Sts.Unit.cmd_Start )
      Contact( "EM00".PackML_Sts.Unit.moduleActive )
   END_RUNG wire#w1
   RUNG wire#powerrail
      Contact( "EM01".PackML_Sts.Unit.cmd_Start )
      Contact( "EM01".PackML_Sts.Unit.moduleActive )
   END_RUNG wire#w1
   RUNG wire#powerrail
      Contact( "EM02".PackML_Sts.Unit.cmd_Start )
      Contact( "EM02".PackML_Sts.Unit.moduleActive )
   END_RUNG wire#w1
   // the same network as SCL:
   "UN".PackML_Sts.cmd_Start := ("UN".PackML_Sts_Alarm.cmd_Start AND "UN".PackML_Sts_Alarm.moduleActive) OR ("EM00".PackML_Sts.Unit.cmd_Start AND "EM00".PackML_Sts.Unit.moduleActive) OR ("EM01".PackML_Sts.Unit.cmd_Start AND "EM01".PackML_Sts.Unit.moduleActive) OR ("EM02".PackML_Sts.Unit.cmd_Start AND "EM02".PackML_Sts.Unit.moduleActive);
END_REGION

REGION Network 4: UN - Starting State Complete
   RUNG wire#powerrail
      Contact( "UN".PackML_Sts_Alarm.sts_Starting_SC )
      wire#w1
      Contact( "EM00".PackML_Sts.Unit.sts_Starting_SC )
      wire#w2
      Contact( "EM01".PackML_Sts.Unit.sts_Starting_SC )
      wire#w3
      Contact( "EM02".PackML_Sts.Unit.sts_Starting_SC )
      wire#w4
      Coil( "UN".PackML_Sts.sts_Starting_SC )
   END_RUNG
   RUNG wire#powerrail
      I_Contact( "UN".PackML_Sts_Alarm.moduleActive )
   END_RUNG wire#w1
   RUNG wire#w1
      I_Contact( "EM00".PackML_Sts.Unit.moduleActive )
   END_RUNG wire#w2
   RUNG wire#w2
      I_Contact( "EM01".PackML_Sts.Unit.moduleActive )
   END_RUNG wire#w3
   RUNG wire#w3
      I_Contact( "EM02".PackML_Sts.Unit.moduleActive )
   END_RUNG wire#w4
   // the same network as SCL:
   "UN".PackML_Sts.sts_Starting_SC := ("UN".PackML_Sts_Alarm.sts_Starting_SC OR NOT "UN".PackML_Sts_Alarm.moduleActive) AND ("EM00".PackML_Sts.Unit.sts_Starting_SC OR NOT "EM00".PackML_Sts.Unit.moduleActive) AND ("EM01".PackML_Sts.Unit.sts_Starting_SC OR NOT "EM01".PackML_Sts.Unit.moduleActive) AND ("EM02".PackML_Sts.Unit.sts_Starting_SC OR NOT "EM02".PackML_Sts.Unit.moduleActive);
END_REGION

REGION Network 5: UN - Stop Command
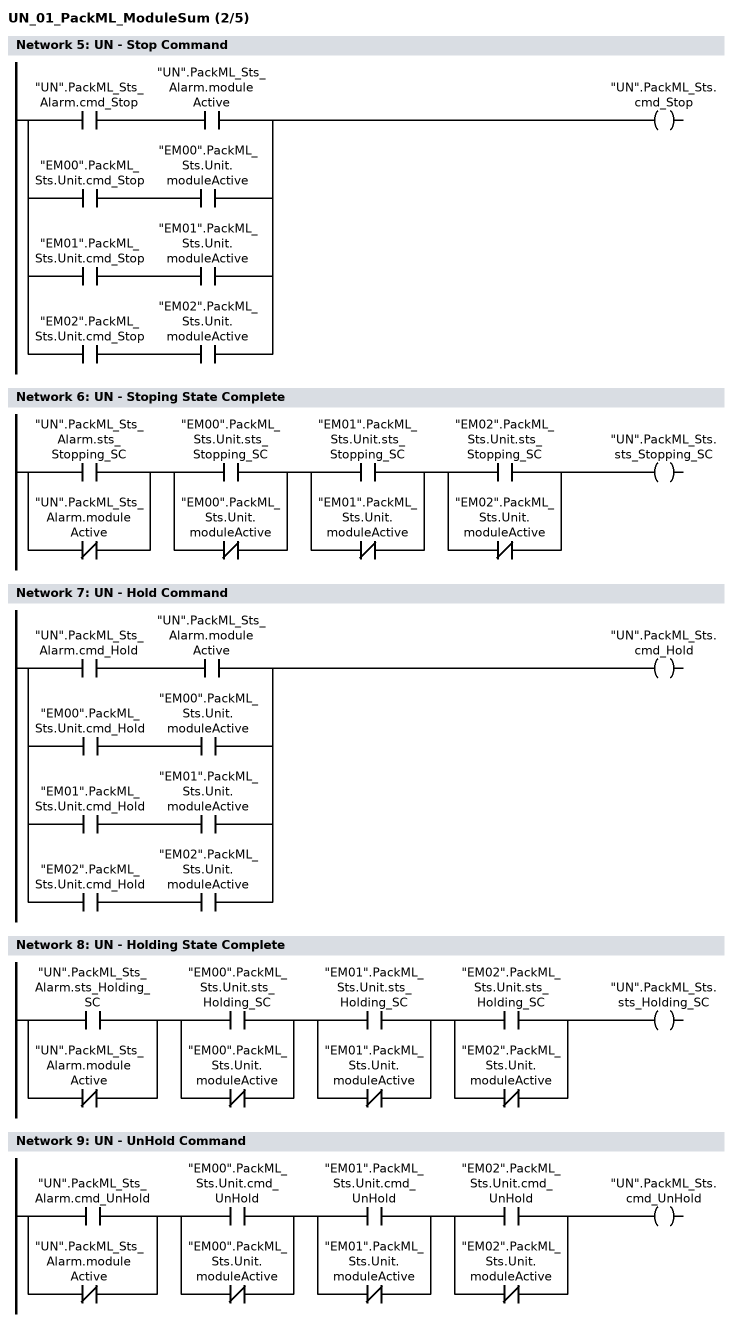
   RUNG wire#powerrail
      Contact( "UN".PackML_Sts_Alarm.cmd_Stop )
      Contact( "UN".PackML_Sts_Alarm.moduleActive )
      wire#w1
      Coil( "UN".PackML_Sts.cmd_Stop )
   END_RUNG
   RUNG wire#powerrail
      Contact( "EM00".PackML_Sts.Unit.cmd_Stop )
      Contact( "EM00".PackML_Sts.Unit.moduleActive )
   END_RUNG wire#w1
   RUNG wire#powerrail
      Contact( "EM01".PackML_Sts.Unit.cmd_Stop )
      Contact( "EM01".PackML_Sts.Unit.moduleActive )
   END_RUNG wire#w1
   RUNG wire#powerrail
      Contact( "EM02".PackML_Sts.Unit.cmd_Stop )
      Contact( "EM02".PackML_Sts.Unit.moduleActive )
   END_RUNG wire#w1
   // the same network as SCL:
   "UN".PackML_Sts.cmd_Stop := ("UN".PackML_Sts_Alarm.cmd_Stop AND "UN".PackML_Sts_Alarm.moduleActive) OR ("EM00".PackML_Sts.Unit.cmd_Stop AND "EM00".PackML_Sts.Unit.moduleActive) OR ("EM01".PackML_Sts.Unit.cmd_Stop AND "EM01".PackML_Sts.Unit.moduleActive) OR ("EM02".PackML_Sts.Unit.cmd_Stop AND "EM02".PackML_Sts.Unit.moduleActive);
END_REGION

REGION Network 6: UN - Stoping State Complete
   RUNG wire#powerrail
      Contact( "UN".PackML_Sts_Alarm.sts_Stopping_SC )
      wire#w1
      Contact( "EM00".PackML_Sts.Unit.sts_Stopping_SC )
      wire#w2
      Contact( "EM01".PackML_Sts.Unit.sts_Stopping_SC )
      wire#w3
      Contact( "EM02".PackML_Sts.Unit.sts_Stopping_SC )
      wire#w4
      Coil( "UN".PackML_Sts.sts_Stopping_SC )
   END_RUNG
   RUNG wire#powerrail
      I_Contact( "UN".PackML_Sts_Alarm.moduleActive )
   END_RUNG wire#w1
   RUNG wire#w1
      I_Contact( "EM00".PackML_Sts.Unit.moduleActive )
   END_RUNG wire#w2
   RUNG wire#w2
      I_Contact( "EM01".PackML_Sts.Unit.moduleActive )
   END_RUNG wire#w3
   RUNG wire#w3
      I_Contact( "EM02".PackML_Sts.Unit.moduleActive )
   END_RUNG wire#w4
   // the same network as SCL:
   "UN".PackML_Sts.sts_Stopping_SC := ("UN".PackML_Sts_Alarm.sts_Stopping_SC OR NOT "UN".PackML_Sts_Alarm.moduleActive) AND ("EM00".PackML_Sts.Unit.sts_Stopping_SC OR NOT "EM00".PackML_Sts.Unit.moduleActive) AND ("EM01".PackML_Sts.Unit.sts_Stopping_SC OR NOT "EM01".PackML_Sts.Unit.moduleActive) AND ("EM02".PackML_Sts.Unit.sts_Stopping_SC OR NOT "EM02".PackML_Sts.Unit.moduleActive);
END_REGION

REGION Network 7: UN - Hold Command
   RUNG wire#powerrail
      Contact( "UN".PackML_Sts_Alarm.cmd_Hold )
      Contact( "UN".PackML_Sts_Alarm.moduleActive )
      wire#w1
      Coil( "UN".PackML_Sts.cmd_Hold )
   END_RUNG
   RUNG wire#powerrail
      Contact( "EM00".PackML_Sts.Unit.cmd_Hold )
      Contact( "EM00".PackML_Sts.Unit.moduleActive )
   END_RUNG wire#w1
   RUNG wire#powerrail
      Contact( "EM01".PackML_Sts.Unit.cmd_Hold )
      Contact( "EM01".PackML_Sts.Unit.moduleActive )
   END_RUNG wire#w1
   RUNG wire#powerrail
      Contact( "EM02".PackML_Sts.Unit.cmd_Hold )
      Contact( "EM02".PackML_Sts.Unit.moduleActive )
   END_RUNG wire#w1
   // the same network as SCL:
   "UN".PackML_Sts.cmd_Hold := ("UN".PackML_Sts_Alarm.cmd_Hold AND "UN".PackML_Sts_Alarm.moduleActive) OR ("EM00".PackML_Sts.Unit.cmd_Hold AND "EM00".PackML_Sts.Unit.moduleActive) OR ("EM01".PackML_Sts.Unit.cmd_Hold AND "EM01".PackML_Sts.Unit.moduleActive) OR ("EM02".PackML_Sts.Unit.cmd_Hold AND "EM02".PackML_Sts.Unit.moduleActive);
END_REGION

REGION Network 8: UN - Holding State Complete
   RUNG wire#powerrail
      Contact( "UN".PackML_Sts_Alarm.sts_Holding_SC )
      wire#w1
      Contact( "EM00".PackML_Sts.Unit.sts_Holding_SC )
      wire#w2
      Contact( "EM01".PackML_Sts.Unit.sts_Holding_SC )
      wire#w3
      Contact( "EM02".PackML_Sts.Unit.sts_Holding_SC )
      wire#w4
      Coil( "UN".PackML_Sts.sts_Holding_SC )
   END_RUNG
   RUNG wire#powerrail
      I_Contact( "UN".PackML_Sts_Alarm.moduleActive )
   END_RUNG wire#w1
   RUNG wire#w1
      I_Contact( "EM00".PackML_Sts.Unit.moduleActive )
   END_RUNG wire#w2
   RUNG wire#w2
      I_Contact( "EM01".PackML_Sts.Unit.moduleActive )
   END_RUNG wire#w3
   RUNG wire#w3
      I_Contact( "EM02".PackML_Sts.Unit.moduleActive )
   END_RUNG wire#w4
   // the same network as SCL:
   "UN".PackML_Sts.sts_Holding_SC := ("UN".PackML_Sts_Alarm.sts_Holding_SC OR NOT "UN".PackML_Sts_Alarm.moduleActive) AND ("EM00".PackML_Sts.Unit.sts_Holding_SC OR NOT "EM00".PackML_Sts.Unit.moduleActive) AND ("EM01".PackML_Sts.Unit.sts_Holding_SC OR NOT "EM01".PackML_Sts.Unit.moduleActive) AND ("EM02".PackML_Sts.Unit.sts_Holding_SC OR NOT "EM02".PackML_Sts.Unit.moduleActive);
END_REGION

REGION Network 9: UN - UnHold Command
   RUNG wire#powerrail
      Contact( "UN".PackML_Sts_Alarm.cmd_UnHold )
      wire#w1
      Contact( "EM00".PackML_Sts.Unit.cmd_UnHold )
      wire#w2
      Contact( "EM01".PackML_Sts.Unit.cmd_UnHold )
      wire#w3
      Contact( "EM02".PackML_Sts.Unit.cmd_UnHold )
      wire#w4
      Coil( "UN".PackML_Sts.cmd_UnHold )
   END_RUNG
   RUNG wire#powerrail
      I_Contact( "UN".PackML_Sts_Alarm.moduleActive )
   END_RUNG wire#w1
   RUNG wire#w1
      I_Contact( "EM00".PackML_Sts.Unit.moduleActive )
   END_RUNG wire#w2
   RUNG wire#w2
      I_Contact( "EM01".PackML_Sts.Unit.moduleActive )
   END_RUNG wire#w3
   RUNG wire#w3
      I_Contact( "EM02".PackML_Sts.Unit.moduleActive )
   END_RUNG wire#w4
   // the same network as SCL:
   "UN".PackML_Sts.cmd_UnHold := ("UN".PackML_Sts_Alarm.cmd_UnHold OR NOT "UN".PackML_Sts_Alarm.moduleActive) AND ("EM00".PackML_Sts.Unit.cmd_UnHold OR NOT "EM00".PackML_Sts.Unit.moduleActive) AND ("EM01".PackML_Sts.Unit.cmd_UnHold OR NOT "EM01".PackML_Sts.Unit.moduleActive) AND ("EM02".PackML_Sts.Unit.cmd_UnHold OR NOT "EM02".PackML_Sts.Unit.moduleActive);
END_REGION

REGION Network 10: UN - UnHolding State Complete
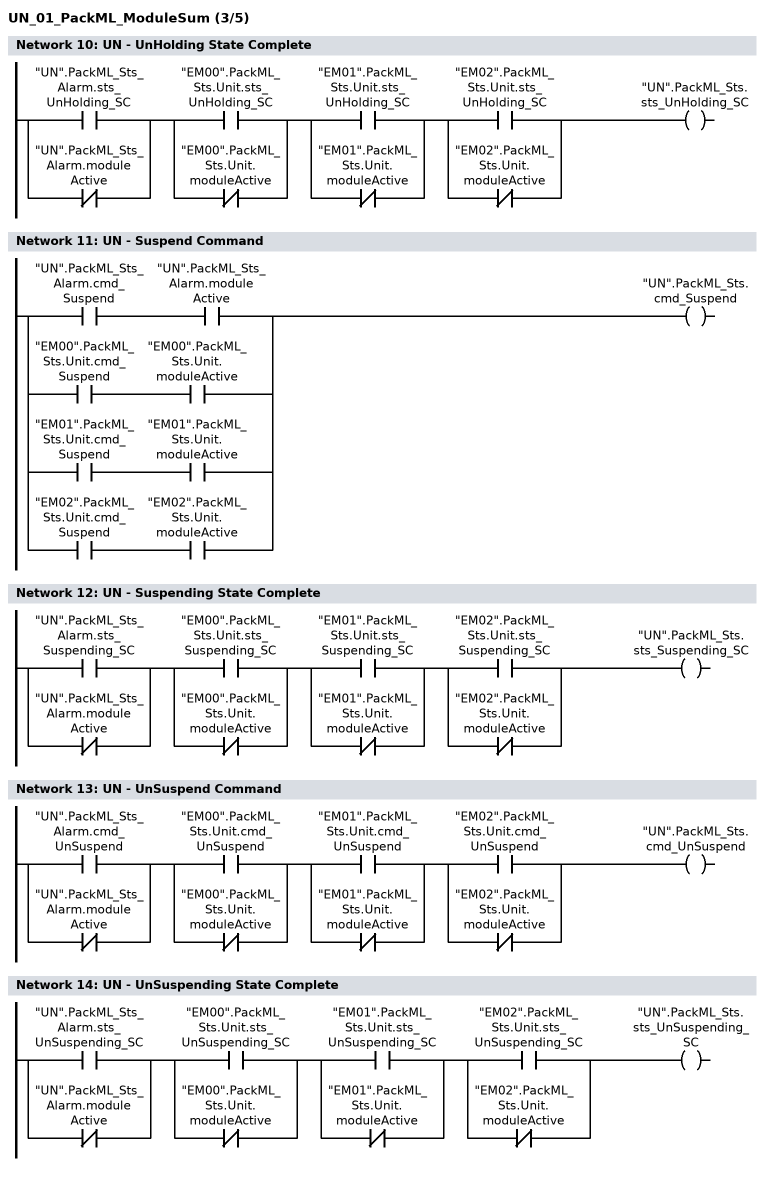
   RUNG wire#powerrail
      Contact( "UN".PackML_Sts_Alarm.sts_UnHolding_SC )
      wire#w1
      Contact( "EM00".PackML_Sts.Unit.sts_UnHolding_SC )
      wire#w2
      Contact( "EM01".PackML_Sts.Unit.sts_UnHolding_SC )
      wire#w3
      Contact( "EM02".PackML_Sts.Unit.sts_UnHolding_SC )
      wire#w4
      Coil( "UN".PackML_Sts.sts_UnHolding_SC )
   END_RUNG
   RUNG wire#powerrail
      I_Contact( "UN".PackML_Sts_Alarm.moduleActive )
   END_RUNG wire#w1
   RUNG wire#w1
      I_Contact( "EM00".PackML_Sts.Unit.moduleActive )
   END_RUNG wire#w2
   RUNG wire#w2
      I_Contact( "EM01".PackML_Sts.Unit.moduleActive )
   END_RUNG wire#w3
   RUNG wire#w3
      I_Contact( "EM02".PackML_Sts.Unit.moduleActive )
   END_RUNG wire#w4
   // the same network as SCL:
   "UN".PackML_Sts.sts_UnHolding_SC := ("UN".PackML_Sts_Alarm.sts_UnHolding_SC OR NOT "UN".PackML_Sts_Alarm.moduleActive) AND ("EM00".PackML_Sts.Unit.sts_UnHolding_SC OR NOT "EM00".PackML_Sts.Unit.moduleActive) AND ("EM01".PackML_Sts.Unit.sts_UnHolding_SC OR NOT "EM01".PackML_Sts.Unit.moduleActive) AND ("EM02".PackML_Sts.Unit.sts_UnHolding_SC OR NOT "EM02".PackML_Sts.Unit.moduleActive);
END_REGION

REGION Network 11: UN - Suspend Command
   RUNG wire#powerrail
      Contact( "UN".PackML_Sts_Alarm.cmd_Suspend )
      Contact( "UN".PackML_Sts_Alarm.moduleActive )
      wire#w1
      Coil( "UN".PackML_Sts.cmd_Suspend )
   END_RUNG
   RUNG wire#powerrail
      Contact( "EM00".PackML_Sts.Unit.cmd_Suspend )
      Contact( "EM00".PackML_Sts.Unit.moduleActive )
   END_RUNG wire#w1
   RUNG wire#powerrail
      Contact( "EM01".PackML_Sts.Unit.cmd_Suspend )
      Contact( "EM01".PackML_Sts.Unit.moduleActive )
   END_RUNG wire#w1
   RUNG wire#powerrail
      Contact( "EM02".PackML_Sts.Unit.cmd_Suspend )
      Contact( "EM02".PackML_Sts.Unit.moduleActive )
   END_RUNG wire#w1
   // the same network as SCL:
   "UN".PackML_Sts.cmd_Suspend := ("UN".PackML_Sts_Alarm.cmd_Suspend AND "UN".PackML_Sts_Alarm.moduleActive) OR ("EM00".PackML_Sts.Unit.cmd_Suspend AND "EM00".PackML_Sts.Unit.moduleActive) OR ("EM01".PackML_Sts.Unit.cmd_Suspend AND "EM01".PackML_Sts.Unit.moduleActive) OR ("EM02".PackML_Sts.Unit.cmd_Suspend AND "EM02".PackML_Sts.Unit.moduleActive);
END_REGION

REGION Network 12: UN - Suspending State Complete
   RUNG wire#powerrail
      Contact( "UN".PackML_Sts_Alarm.sts_Suspending_SC )
      wire#w1
      Contact( "EM00".PackML_Sts.Unit.sts_Suspending_SC )
      wire#w2
      Contact( "EM01".PackML_Sts.Unit.sts_Suspending_SC )
      wire#w3
      Contact( "EM02".PackML_Sts.Unit.sts_Suspending_SC )
      wire#w4
      Coil( "UN".PackML_Sts.sts_Suspending_SC )
   END_RUNG
   RUNG wire#powerrail
      I_Contact( "UN".PackML_Sts_Alarm.moduleActive )
   END_RUNG wire#w1
   RUNG wire#w1
      I_Contact( "EM00".PackML_Sts.Unit.moduleActive )
   END_RUNG wire#w2
   RUNG wire#w2
      I_Contact( "EM01".PackML_Sts.Unit.moduleActive )
   END_RUNG wire#w3
   RUNG wire#w3
      I_Contact( "EM02".PackML_Sts.Unit.moduleActive )
   END_RUNG wire#w4
   // the same network as SCL:
   "UN".PackML_Sts.sts_Suspending_SC := ("UN".PackML_Sts_Alarm.sts_Suspending_SC OR NOT "UN".PackML_Sts_Alarm.moduleActive) AND ("EM00".PackML_Sts.Unit.sts_Suspending_SC OR NOT "EM00".PackML_Sts.Unit.moduleActive) AND ("EM01".PackML_Sts.Unit.sts_Suspending_SC OR NOT "EM01".PackML_Sts.Unit.moduleActive) AND ("EM02".PackML_Sts.Unit.sts_Suspending_SC OR NOT "EM02".PackML_Sts.Unit.moduleActive);
END_REGION

REGION Network 13: UN - UnSuspend Command
   RUNG wire#powerrail
      Contact( "UN".PackML_Sts_Alarm.cmd_UnSuspend )
      wire#w1
      Contact( "EM00".PackML_Sts.Unit.cmd_UnSuspend )
      wire#w2
      Contact( "EM01".PackML_Sts.Unit.cmd_UnSuspend )
      wire#w3
      Contact( "EM02".PackML_Sts.Unit.cmd_UnSuspend )
      wire#w4
      Coil( "UN".PackML_Sts.cmd_UnSuspend )
   END_RUNG
   RUNG wire#powerrail
      I_Contact( "UN".PackML_Sts_Alarm.moduleActive )
   END_RUNG wire#w1
   RUNG wire#w1
      I_Contact( "EM00".PackML_Sts.Unit.moduleActive )
   END_RUNG wire#w2
   RUNG wire#w2
      I_Contact( "EM01".PackML_Sts.Unit.moduleActive )
   END_RUNG wire#w3
   RUNG wire#w3
      I_Contact( "EM02".PackML_Sts.Unit.moduleActive )
   END_RUNG wire#w4
   // the same network as SCL:
   "UN".PackML_Sts.cmd_UnSuspend := ("UN".PackML_Sts_Alarm.cmd_UnSuspend OR NOT "UN".PackML_Sts_Alarm.moduleActive) AND ("EM00".PackML_Sts.Unit.cmd_UnSuspend OR NOT "EM00".PackML_Sts.Unit.moduleActive) AND ("EM01".PackML_Sts.Unit.cmd_UnSuspend OR NOT "EM01".PackML_Sts.Unit.moduleActive) AND ("EM02".PackML_Sts.Unit.cmd_UnSuspend OR NOT "EM02".PackML_Sts.Unit.moduleActive);
END_REGION

REGION Network 14: UN - UnSuspending State Complete
   RUNG wire#powerrail
      Contact( "UN".PackML_Sts_Alarm.sts_UnSuspending_SC )
      wire#w1
      Contact( "EM00".PackML_Sts.Unit.sts_UnSuspending_SC )
      wire#w2
      Contact( "EM01".PackML_Sts.Unit.sts_UnSuspending_SC )
      wire#w3
      Contact( "EM02".PackML_Sts.Unit.sts_UnSuspending_SC )
      wire#w4
      Coil( "UN".PackML_Sts.sts_UnSuspending_SC )
   END_RUNG
   RUNG wire#powerrail
      I_Contact( "UN".PackML_Sts_Alarm.moduleActive )
   END_RUNG wire#w1
   RUNG wire#w1
      I_Contact( "EM00".PackML_Sts.Unit.moduleActive )
   END_RUNG wire#w2
   RUNG wire#w2
      I_Contact( "EM01".PackML_Sts.Unit.moduleActive )
   END_RUNG wire#w3
   RUNG wire#w3
      I_Contact( "EM02".PackML_Sts.Unit.moduleActive )
   END_RUNG wire#w4
   // the same network as SCL:
   "UN".PackML_Sts.sts_UnSuspending_SC := ("UN".PackML_Sts_Alarm.sts_UnSuspending_SC OR NOT "UN".PackML_Sts_Alarm.moduleActive) AND ("EM00".PackML_Sts.Unit.sts_UnSuspending_SC OR NOT "EM00".PackML_Sts.Unit.moduleActive) AND ("EM01".PackML_Sts.Unit.sts_UnSuspending_SC OR NOT "EM01".PackML_Sts.Unit.moduleActive) AND ("EM02".PackML_Sts.Unit.sts_UnSuspending_SC OR NOT "EM02".PackML_Sts.Unit.moduleActive);
END_REGION

REGION Network 15: UN - Abort Command
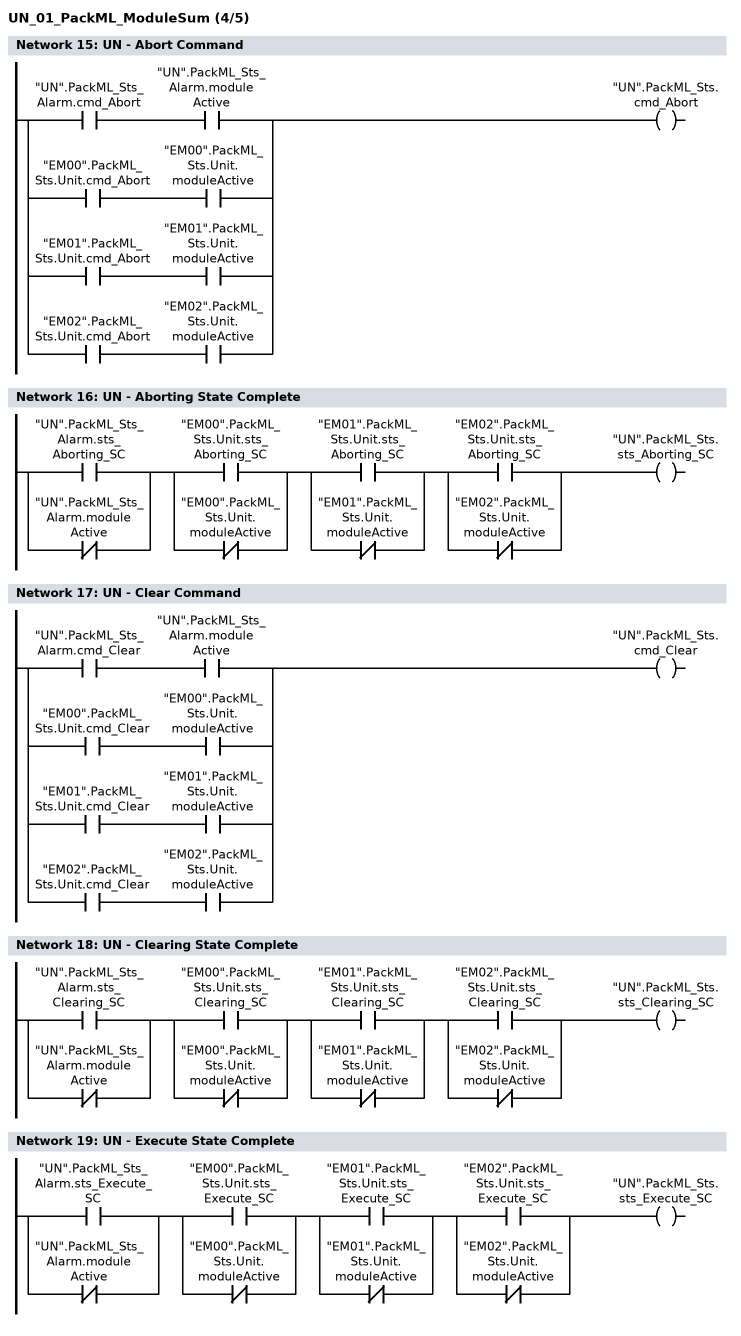
   RUNG wire#powerrail
      Contact( "UN".PackML_Sts_Alarm.cmd_Abort )
      Contact( "UN".PackML_Sts_Alarm.moduleActive )
      wire#w1
      Coil( "UN".PackML_Sts.cmd_Abort )
   END_RUNG
   RUNG wire#powerrail
      Contact( "EM00".PackML_Sts.Unit.cmd_Abort )
      Contact( "EM00".PackML_Sts.Unit.moduleActive )
   END_RUNG wire#w1
   RUNG wire#powerrail
      Contact( "EM01".PackML_Sts.Unit.cmd_Abort )
      Contact( "EM01".PackML_Sts.Unit.moduleActive )
   END_RUNG wire#w1
   RUNG wire#powerrail
      Contact( "EM02".PackML_Sts.Unit.cmd_Abort )
      Contact( "EM02".PackML_Sts.Unit.moduleActive )
   END_RUNG wire#w1
   // the same network as SCL:
   "UN".PackML_Sts.cmd_Abort := ("UN".PackML_Sts_Alarm.cmd_Abort AND "UN".PackML_Sts_Alarm.moduleActive) OR ("EM00".PackML_Sts.Unit.cmd_Abort AND "EM00".PackML_Sts.Unit.moduleActive) OR ("EM01".PackML_Sts.Unit.cmd_Abort AND "EM01".PackML_Sts.Unit.moduleActive) OR ("EM02".PackML_Sts.Unit.cmd_Abort AND "EM02".PackML_Sts.Unit.moduleActive);
END_REGION

REGION Network 16: UN - Aborting State Complete
   RUNG wire#powerrail
      Contact( "UN".PackML_Sts_Alarm.sts_Aborting_SC )
      wire#w1
      Contact( "EM00".PackML_Sts.Unit.sts_Aborting_SC )
      wire#w2
      Contact( "EM01".PackML_Sts.Unit.sts_Aborting_SC )
      wire#w3
      Contact( "EM02".PackML_Sts.Unit.sts_Aborting_SC )
      wire#w4
      Coil( "UN".PackML_Sts.sts_Aborting_SC )
   END_RUNG
   RUNG wire#powerrail
      I_Contact( "UN".PackML_Sts_Alarm.moduleActive )
   END_RUNG wire#w1
   RUNG wire#w1
      I_Contact( "EM00".PackML_Sts.Unit.moduleActive )
   END_RUNG wire#w2
   RUNG wire#w2
      I_Contact( "EM01".PackML_Sts.Unit.moduleActive )
   END_RUNG wire#w3
   RUNG wire#w3
      I_Contact( "EM02".PackML_Sts.Unit.moduleActive )
   END_RUNG wire#w4
   // the same network as SCL:
   "UN".PackML_Sts.sts_Aborting_SC := ("UN".PackML_Sts_Alarm.sts_Aborting_SC OR NOT "UN".PackML_Sts_Alarm.moduleActive) AND ("EM00".PackML_Sts.Unit.sts_Aborting_SC OR NOT "EM00".PackML_Sts.Unit.moduleActive) AND ("EM01".PackML_Sts.Unit.sts_Aborting_SC OR NOT "EM01".PackML_Sts.Unit.moduleActive) AND ("EM02".PackML_Sts.Unit.sts_Aborting_SC OR NOT "EM02".PackML_Sts.Unit.moduleActive);
END_REGION

REGION Network 17: UN - Clear Command
   RUNG wire#powerrail
      Contact( "UN".PackML_Sts_Alarm.cmd_Clear )
      Contact( "UN".PackML_Sts_Alarm.moduleActive )
      wire#w1
      Coil( "UN".PackML_Sts.cmd_Clear )
   END_RUNG
   RUNG wire#powerrail
      Contact( "EM00".PackML_Sts.Unit.cmd_Clear )
      Contact( "EM00".PackML_Sts.Unit.moduleActive )
   END_RUNG wire#w1
   RUNG wire#powerrail
      Contact( "EM01".PackML_Sts.Unit.cmd_Clear )
      Contact( "EM01".PackML_Sts.Unit.moduleActive )
   END_RUNG wire#w1
   RUNG wire#powerrail
      Contact( "EM02".PackML_Sts.Unit.cmd_Clear )
      Contact( "EM02".PackML_Sts.Unit.moduleActive )
   END_RUNG wire#w1
   // the same network as SCL:
   "UN".PackML_Sts.cmd_Clear := ("UN".PackML_Sts_Alarm.cmd_Clear AND "UN".PackML_Sts_Alarm.moduleActive) OR ("EM00".PackML_Sts.Unit.cmd_Clear AND "EM00".PackML_Sts.Unit.moduleActive) OR ("EM01".PackML_Sts.Unit.cmd_Clear AND "EM01".PackML_Sts.Unit.moduleActive) OR ("EM02".PackML_Sts.Unit.cmd_Clear AND "EM02".PackML_Sts.Unit.moduleActive);
END_REGION

REGION Network 18: UN - Clearing State Complete
   RUNG wire#powerrail
      Contact( "UN".PackML_Sts_Alarm.sts_Clearing_SC )
      wire#w1
      Contact( "EM00".PackML_Sts.Unit.sts_Clearing_SC )
      wire#w2
      Contact( "EM01".PackML_Sts.Unit.sts_Clearing_SC )
      wire#w3
      Contact( "EM02".PackML_Sts.Unit.sts_Clearing_SC )
      wire#w4
      Coil( "UN".PackML_Sts.sts_Clearing_SC )
   END_RUNG
   RUNG wire#powerrail
      I_Contact( "UN".PackML_Sts_Alarm.moduleActive )
   END_RUNG wire#w1
   RUNG wire#w1
      I_Contact( "EM00".PackML_Sts.Unit.moduleActive )
   END_RUNG wire#w2
   RUNG wire#w2
      I_Contact( "EM01".PackML_Sts.Unit.moduleActive )
   END_RUNG wire#w3
   RUNG wire#w3
      I_Contact( "EM02".PackML_Sts.Unit.moduleActive )
   END_RUNG wire#w4
   // the same network as SCL:
   "UN".PackML_Sts.sts_Clearing_SC := ("UN".PackML_Sts_Alarm.sts_Clearing_SC OR NOT "UN".PackML_Sts_Alarm.moduleActive) AND ("EM00".PackML_Sts.Unit.sts_Clearing_SC OR NOT "EM00".PackML_Sts.Unit.moduleActive) AND ("EM01".PackML_Sts.Unit.sts_Clearing_SC OR NOT "EM01".PackML_Sts.Unit.moduleActive) AND ("EM02".PackML_Sts.Unit.sts_Clearing_SC OR NOT "EM02".PackML_Sts.Unit.moduleActive);
END_REGION

REGION Network 19: UN - Execute State Complete
   RUNG wire#powerrail
      Contact( "UN".PackML_Sts_Alarm.sts_Execute_SC )
      wire#w1
      Contact( "EM00".PackML_Sts.Unit.sts_Execute_SC )
      wire#w2
      Contact( "EM01".PackML_Sts.Unit.sts_Execute_SC )
      wire#w3
      Contact( "EM02".PackML_Sts.Unit.sts_Execute_SC )
      wire#w4
      Coil( "UN".PackML_Sts.sts_Execute_SC )
   END_RUNG
   RUNG wire#powerrail
      I_Contact( "UN".PackML_Sts_Alarm.moduleActive )
   END_RUNG wire#w1
   RUNG wire#w1
      I_Contact( "EM00".PackML_Sts.Unit.moduleActive )
   END_RUNG wire#w2
   RUNG wire#w2
      I_Contact( "EM01".PackML_Sts.Unit.moduleActive )
   END_RUNG wire#w3
   RUNG wire#w3
      I_Contact( "EM02".PackML_Sts.Unit.moduleActive )
   END_RUNG wire#w4
   // the same network as SCL:
   "UN".PackML_Sts.sts_Execute_SC := ("UN".PackML_Sts_Alarm.sts_Execute_SC OR NOT "UN".PackML_Sts_Alarm.moduleActive) AND ("EM00".PackML_Sts.Unit.sts_Execute_SC OR NOT "EM00".PackML_Sts.Unit.moduleActive) AND ("EM01".PackML_Sts.Unit.sts_Execute_SC OR NOT "EM01".PackML_Sts.Unit.moduleActive) AND ("EM02".PackML_Sts.Unit.sts_Execute_SC OR NOT "EM02".PackML_Sts.Unit.moduleActive);
END_REGION

REGION Network 20: UN - Completing State Complete
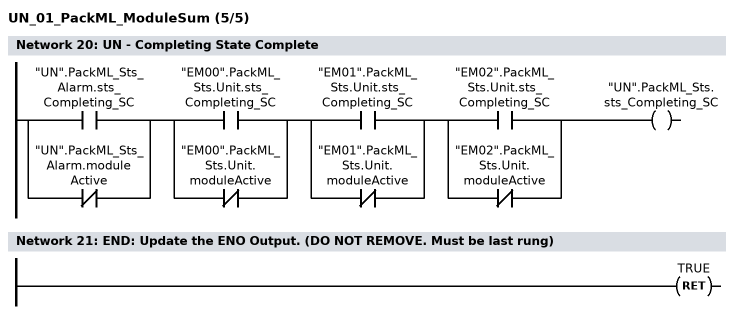
   RUNG wire#powerrail
      Contact( "UN".PackML_Sts_Alarm.sts_Completing_SC )
      wire#w1
      Contact( "EM00".PackML_Sts.Unit.sts_Completing_SC )
      wire#w2
      Contact( "EM01".PackML_Sts.Unit.sts_Completing_SC )
      wire#w3
      Contact( "EM02".PackML_Sts.Unit.sts_Completing_SC )
      wire#w4
      Coil( "UN".PackML_Sts.sts_Completing_SC )
   END_RUNG
   RUNG wire#powerrail
      I_Contact( "UN".PackML_Sts_Alarm.moduleActive )
   END_RUNG wire#w1
   RUNG wire#w1
      I_Contact( "EM00".PackML_Sts.Unit.moduleActive )
   END_RUNG wire#w2
   RUNG wire#w2
      I_Contact( "EM01".PackML_Sts.Unit.moduleActive )
   END_RUNG wire#w3
   RUNG wire#w3
      I_Contact( "EM02".PackML_Sts.Unit.moduleActive )
   END_RUNG wire#w4
   // the same network as SCL:
   "UN".PackML_Sts.sts_Completing_SC := ("UN".PackML_Sts_Alarm.sts_Completing_SC OR NOT "UN".PackML_Sts_Alarm.moduleActive) AND ("EM00".PackML_Sts.Unit.sts_Completing_SC OR NOT "EM00".PackML_Sts.Unit.moduleActive) AND ("EM01".PackML_Sts.Unit.sts_Completing_SC OR NOT "EM01".PackML_Sts.Unit.moduleActive) AND ("EM02".PackML_Sts.Unit.sts_Completing_SC OR NOT "EM02".PackML_Sts.Unit.moduleActive);
END_REGION

REGION Network 21: END: Update the ENO Output. (DO NOT REMOVE. Must be last rung)
   RUNG wire#powerrail
      ReturnCoil( TRUE )
   END_RUNG
   // the same network as SCL:
   ENO := TRUE;
   RETURN;
END_REGION
END_FUNCTION_BLOCK

FUNCTION_BLOCK "UN_02_PackML"   // FB31622, LAD
TITLE = UN_02_PackML
{ S7_Optimized_Access := 'TRUE' }
AUTHOR : tech.team.motioncontrol@siemens.com
FAMILY : CPG
VERSION : 1.0
// Support: tech.team.motioncontrol@siemens.com
// Fax: +49 (0) 9131/98-1297
// stored: AutoNumber true, IsIECCheckEnabled false, IsRetainMemResEnabled false, MemoryReserve 100, SetENOAutomatically false, UDAEnableTagReadback false
   VAR
      statLanguageSelectedOld { ExternalAccessible := 'False'; ExternalVisible := 'False'; ExternalWritable := 'False'} : Int := -1;
      statPackML_CMD_SC { ExternalAccessible := 'False'; ExternalVisible := 'False'; ExternalWritable := 'False'} : Bool;
      instUnitModeStateManager { ExternalAccessible := 'False'; ExternalVisible := 'False'; ExternalWritable := 'False'; S7_SetPoint := 'True'} : "LPMLV30_UnitModeStateManager";
      instUnitModeStateTimes { ExternalAccessible := 'False'; ExternalVisible := 'False'; ExternalWritable := 'False'; S7_SetPoint := 'True'} : "LPMLV30_UnitModeStateTimes";
      statRemoteCommand_ModeChangeRequest { ExternalAccessible := 'False'; ExternalVisible := 'False'; ExternalWritable := 'False'} : Struct
         Production { ExternalAccessible := 'False'; ExternalVisible := 'False'; ExternalWritable := 'False'} : Bool;   // Request to goto mode - PRODUCTION (mode #1)
         Maintenance { ExternalAccessible := 'False'; ExternalVisible := 'False'; ExternalWritable := 'False'} : Bool;   // Request to goto mode - MAINTENANCE (mode #2)
         Manual { ExternalAccessible := 'False'; ExternalVisible := 'False'; ExternalWritable := 'False'} : Bool;   // Request to goto mode - MANUAL (mode #3)
         UserMode01 { ExternalAccessible := 'False'; ExternalVisible := 'False'; ExternalWritable := 'False'} : Bool;   // Request to goto mode - USER MODE 01 (mode #4)
         UserMode02 { ExternalAccessible := 'False'; ExternalVisible := 'False'; ExternalWritable := 'False'} : Bool;   // Request to goto mode - USER MODE 02 (mode #5)
         UserMode03 { ExternalAccessible := 'False'; ExternalVisible := 'False'; ExternalWritable := 'False'} : Bool;   // Request to goto mode - USER MODE 03 (mode #6)
         UserMode04 { ExternalAccessible := 'False'; ExternalVisible := 'False'; ExternalWritable := 'False'} : Bool;   // Request to goto mode - USER MODE 04 (mode #7)
         UserMode05 { ExternalAccessible := 'False'; ExternalVisible := 'False'; ExternalWritable := 'False'} : Bool;   // Request to goto mode - USER MODE 05 (mode #8)
         UserMode06 { ExternalAccessible := 'False'; ExternalVisible := 'False'; ExternalWritable := 'False'} : Bool;   // Request to goto mode - USER MODE 06 (mode #9)
         UserMode07 { ExternalAccessible := 'False'; ExternalVisible := 'False'; ExternalWritable := 'False'} : Bool;   // Request to goto mode - USER MODE 07 (mode #10)
         UserMode08 { ExternalAccessible := 'False'; ExternalVisible := 'False'; ExternalWritable := 'False'} : Bool;   // Request to goto mode - USER MODE 08 (mode #11)
      END_STRUCT;
      TPResettingDelay { ExternalAccessible := 'False'; ExternalVisible := 'False'; ExternalWritable := 'False'; S7_SetPoint := 'True'} : TP_TIME;
      TPClearingDelay { ExternalAccessible := 'False'; ExternalVisible := 'False'; ExternalWritable := 'False'; S7_SetPoint := 'True'} : TP_TIME;
   END_VAR
   VAR_TEMP
      tempDiagnosticsBufferIndexForHMI : Int;   // Temporary integer for PackML HMI diagnostics
   END_VAR
   VAR_TEMP   // added for the SCL form of the ladder/FBD networks
      _w1 : Bool;
   END_VAR
BEGIN

REGION Network 1: PackML ModeManager & State Model - Reset command
   // Reset Command:
   // If the machine is stopped and there are no faults (no stop or abort commands), 
   // then automatically reset and move the machine to idle.  This is common when all 
   // the faults are cleared in the Clearing state and the machine moves to the 
   // Stopped state with no more faults.
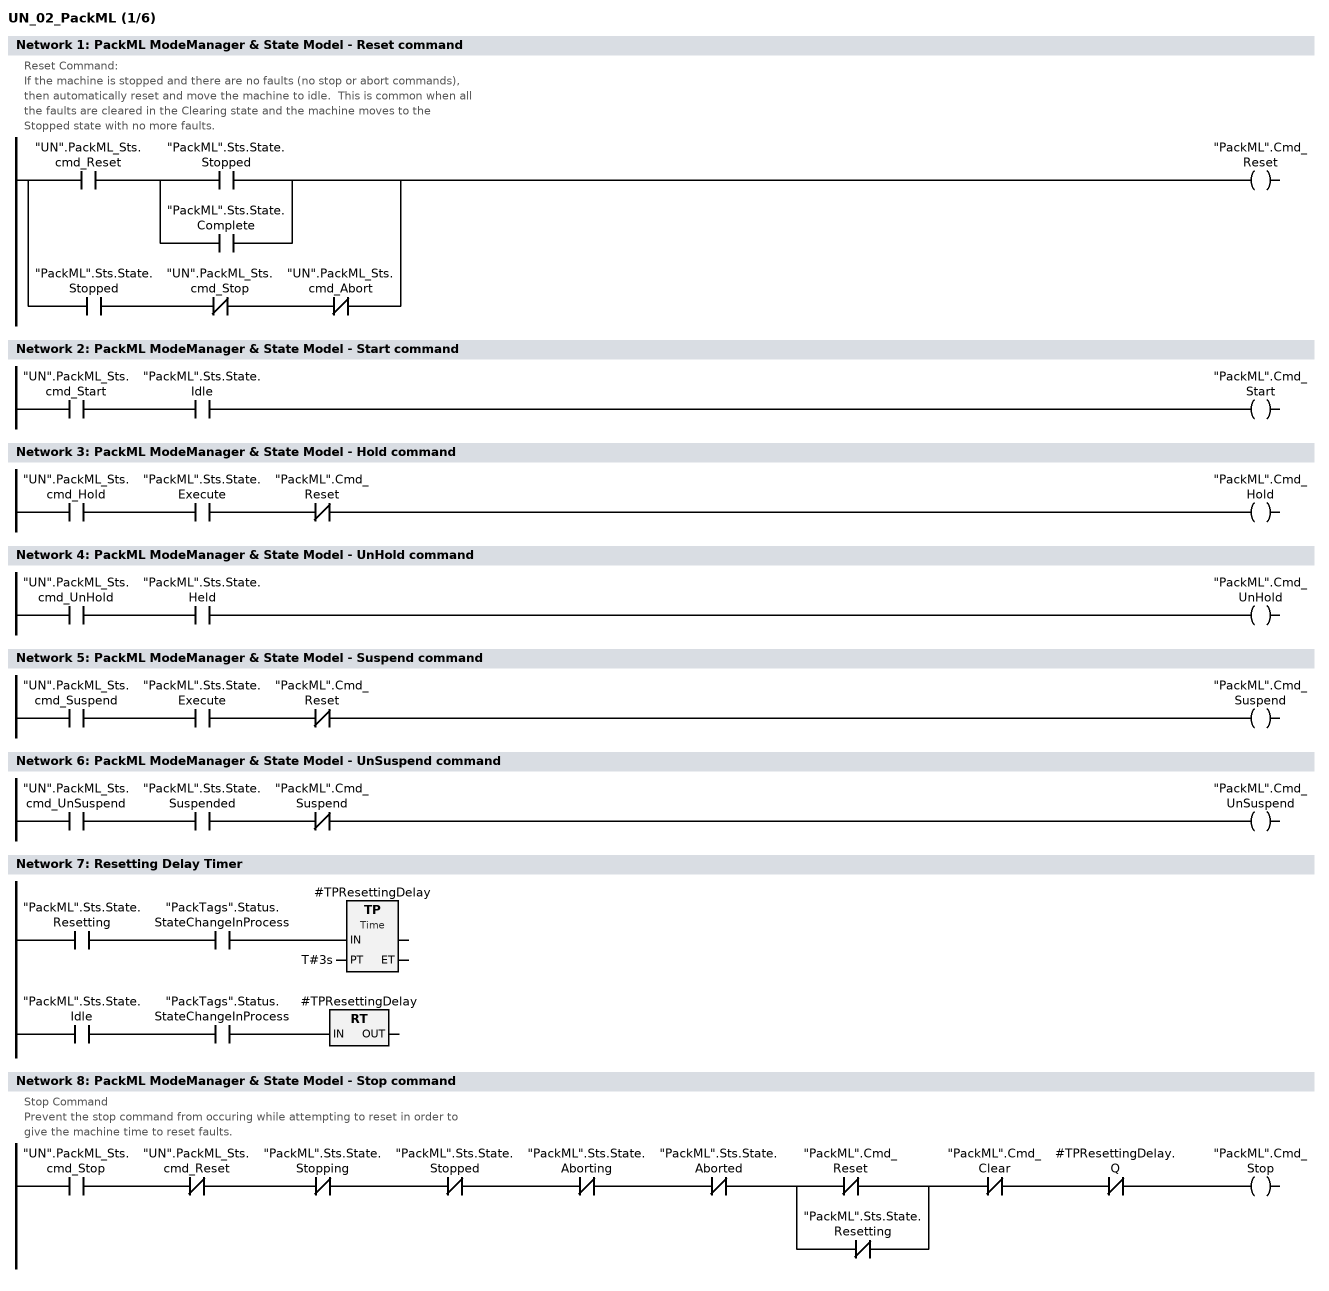
   RUNG wire#powerrail
      Contact( "UN".PackML_Sts.cmd_Reset )
      wire#w1
      Contact( "PackML".Sts.State.Stopped )
      wire#w2
      Coil( "PackML".Cmd_Reset )
   END_RUNG
   RUNG wire#w1
      Contact( "PackML".Sts.State.Complete )
   END_RUNG wire#w2
   RUNG wire#powerrail
      Contact( "PackML".Sts.State.Stopped )
      I_Contact( "UN".PackML_Sts.cmd_Stop )
      I_Contact( "UN".PackML_Sts.cmd_Abort )
   END_RUNG wire#w2
   // the same network as SCL:
   "PackML".Cmd_Reset := ("UN".PackML_Sts.cmd_Reset AND ("PackML".Sts.State.Stopped OR "PackML".Sts.State.Complete)) OR ("PackML".Sts.State.Stopped AND NOT "UN".PackML_Sts.cmd_Stop AND NOT "UN".PackML_Sts.cmd_Abort);
END_REGION

REGION Network 2: PackML ModeManager & State Model - Start command
   RUNG wire#powerrail
      Contact( "UN".PackML_Sts.cmd_Start )
      Contact( "PackML".Sts.State.Idle )
      Coil( "PackML".Cmd_Start )
   END_RUNG
   // the same network as SCL:
   "PackML".Cmd_Start := "UN".PackML_Sts.cmd_Start AND "PackML".Sts.State.Idle;
END_REGION

REGION Network 3: PackML ModeManager & State Model - Hold command
   RUNG wire#powerrail
      Contact( "UN".PackML_Sts.cmd_Hold )
      Contact( "PackML".Sts.State.Execute )
      I_Contact( "PackML".Cmd_Reset )
      Coil( "PackML".Cmd_Hold )
   END_RUNG
   // the same network as SCL:
   "PackML".Cmd_Hold := "UN".PackML_Sts.cmd_Hold AND "PackML".Sts.State.Execute AND NOT "PackML".Cmd_Reset;
END_REGION

REGION Network 4: PackML ModeManager & State Model - UnHold command
   RUNG wire#powerrail
      Contact( "UN".PackML_Sts.cmd_UnHold )
      Contact( "PackML".Sts.State.Held )
      Coil( "PackML".Cmd_UnHold )
   END_RUNG
   // the same network as SCL:
   "PackML".Cmd_UnHold := "UN".PackML_Sts.cmd_UnHold AND "PackML".Sts.State.Held;
END_REGION

REGION Network 5: PackML ModeManager & State Model - Suspend command
   RUNG wire#powerrail
      Contact( "UN".PackML_Sts.cmd_Suspend )
      Contact( "PackML".Sts.State.Execute )
      I_Contact( "PackML".Cmd_Reset )
      Coil( "PackML".Cmd_Suspend )
   END_RUNG
   // the same network as SCL:
   "PackML".Cmd_Suspend := "UN".PackML_Sts.cmd_Suspend AND "PackML".Sts.State.Execute AND NOT "PackML".Cmd_Reset;
END_REGION

REGION Network 6: PackML ModeManager & State Model - UnSuspend command
   RUNG wire#powerrail
      Contact( "UN".PackML_Sts.cmd_UnSuspend )
      Contact( "PackML".Sts.State.Suspended )
      I_Contact( "PackML".Cmd_Suspend )
      Coil( "PackML".Cmd_UnSuspend )
   END_RUNG
   // the same network as SCL:
   "PackML".Cmd_UnSuspend := "UN".PackML_Sts.cmd_UnSuspend AND "PackML".Sts.State.Suspended AND NOT "PackML".Cmd_Suspend;
END_REGION

REGION Network 7: Resetting Delay Timer
   RUNG wire#powerrail
      Contact( "PackML".Sts.State.Resetting )
      Contact( "PackTags".Status.StateChangeInProcess )
      { S7_Templates := "time_type := Time" } #TPResettingDelay.TP(pt := T#3s, et =>)
   END_RUNG
   RUNG wire#powerrail
      Contact( "PackML".Sts.State.Idle )
      Contact( "PackTags".Status.StateChangeInProcess )
      RT_Coil( #TPResettingDelay )
   END_RUNG
   // the same network as SCL:
   #TPResettingDelay(IN := "PackML".Sts.State.Resetting AND "PackTags".Status.StateChangeInProcess, PT := T#3s);   // TP
   IF "PackML".Sts.State.Idle AND "PackTags".Status.StateChangeInProcess THEN
       RESET_TIMER(#TPResettingDelay);
   END_IF;
END_REGION

REGION Network 8: PackML ModeManager & State Model - Stop command
   // Stop Command
   // Prevent the stop command from occuring while attempting to reset in order to 
   // give the machine time to reset faults.
   RUNG wire#powerrail
      Contact( "UN".PackML_Sts.cmd_Stop )
      I_Contact( "UN".PackML_Sts.cmd_Reset )
      I_Contact( "PackML".Sts.State.Stopping )
      I_Contact( "PackML".Sts.State.Stopped )
      I_Contact( "PackML".Sts.State.Aborting )
      I_Contact( "PackML".Sts.State.Aborted )
      wire#w1
      I_Contact( "PackML".Cmd_Reset )
      wire#w2
      I_Contact( "PackML".Cmd_Clear )
      I_Contact( #TPResettingDelay.Q )
      Coil( "PackML".Cmd_Stop )
   END_RUNG
   RUNG wire#w1
      I_Contact( "PackML".Sts.State.Resetting )
   END_RUNG wire#w2
   // the same network as SCL:
   "PackML".Cmd_Stop := "UN".PackML_Sts.cmd_Stop AND NOT "UN".PackML_Sts.cmd_Reset AND NOT "PackML".Sts.State.Stopping AND NOT "PackML".Sts.State.Stopped AND NOT "PackML".Sts.State.Aborting AND NOT "PackML".Sts.State.Aborted AND (NOT "PackML".Cmd_Reset OR NOT "PackML".Sts.State.Resetting) AND NOT "PackML".Cmd_Clear AND NOT #TPResettingDelay.Q;
END_REGION

REGION Network 9: Clearing Delay Timer
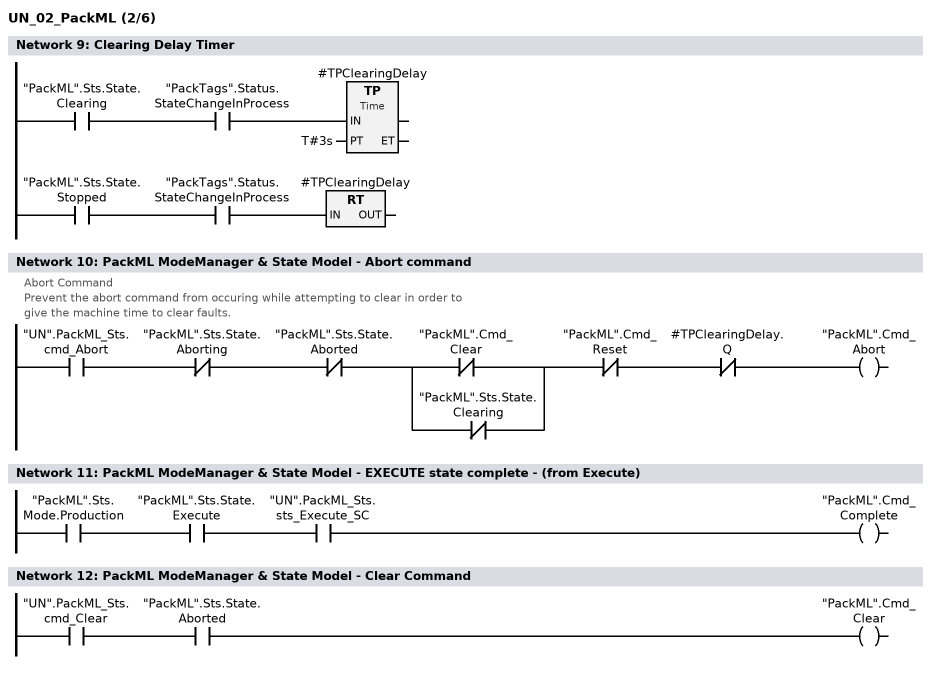
   RUNG wire#powerrail
      Contact( "PackML".Sts.State.Clearing )
      Contact( "PackTags".Status.StateChangeInProcess )
      { S7_Templates := "time_type := Time" } #TPClearingDelay.TP(pt := T#3s, et =>)
   END_RUNG
   RUNG wire#powerrail
      Contact( "PackML".Sts.State.Stopped )
      Contact( "PackTags".Status.StateChangeInProcess )
      RT_Coil( #TPClearingDelay )
   END_RUNG
   // the same network as SCL:
   #TPClearingDelay(IN := "PackML".Sts.State.Clearing AND "PackTags".Status.StateChangeInProcess, PT := T#3s);   // TP
   IF "PackML".Sts.State.Stopped AND "PackTags".Status.StateChangeInProcess THEN
       RESET_TIMER(#TPClearingDelay);
   END_IF;
END_REGION

REGION Network 10: PackML ModeManager & State Model - Abort command
   // Abort Command
   // Prevent the abort command from occuring while attempting to clear in order to 
   // give the machine time to clear faults.
   RUNG wire#powerrail
      Contact( "UN".PackML_Sts.cmd_Abort )
      I_Contact( "PackML".Sts.State.Aborting )
      I_Contact( "PackML".Sts.State.Aborted )
      wire#w1
      I_Contact( "PackML".Cmd_Clear )
      wire#w2
      I_Contact( "PackML".Cmd_Reset )
      I_Contact( #TPClearingDelay.Q )
      Coil( "PackML".Cmd_Abort )
   END_RUNG
   RUNG wire#w1
      I_Contact( "PackML".Sts.State.Clearing )
   END_RUNG wire#w2
   // the same network as SCL:
   "PackML".Cmd_Abort := "UN".PackML_Sts.cmd_Abort AND NOT "PackML".Sts.State.Aborting AND NOT "PackML".Sts.State.Aborted AND (NOT "PackML".Cmd_Clear OR NOT "PackML".Sts.State.Clearing) AND NOT "PackML".Cmd_Reset AND NOT #TPClearingDelay.Q;
END_REGION

REGION Network 11: PackML ModeManager & State Model - EXECUTE state complete - (from Execute)
   RUNG wire#powerrail
      Contact( "PackML".Sts.Mode.Production )
      Contact( "PackML".Sts.State.Execute )
      Contact( "UN".PackML_Sts.sts_Execute_SC )
      Coil( "PackML".Cmd_Complete )
   END_RUNG
   // the same network as SCL:
   "PackML".Cmd_Complete := "PackML".Sts.Mode.Production AND "PackML".Sts.State.Execute AND "UN".PackML_Sts.sts_Execute_SC;
END_REGION

REGION Network 12: PackML ModeManager & State Model - Clear Command
   RUNG wire#powerrail
      Contact( "UN".PackML_Sts.cmd_Clear )
      Contact( "PackML".Sts.State.Aborted )
      Coil( "PackML".Cmd_Clear )
   END_RUNG
   // the same network as SCL:
   "PackML".Cmd_Clear := "UN".PackML_Sts.cmd_Clear AND "PackML".Sts.State.Aborted;
END_REGION

REGION Network 13: External PackML Mode Commands
   // External State Commands are handled in the UN_05_EventControl routine to ensure that the unit machine level alarm manager captures the reason for any machine stoppage.
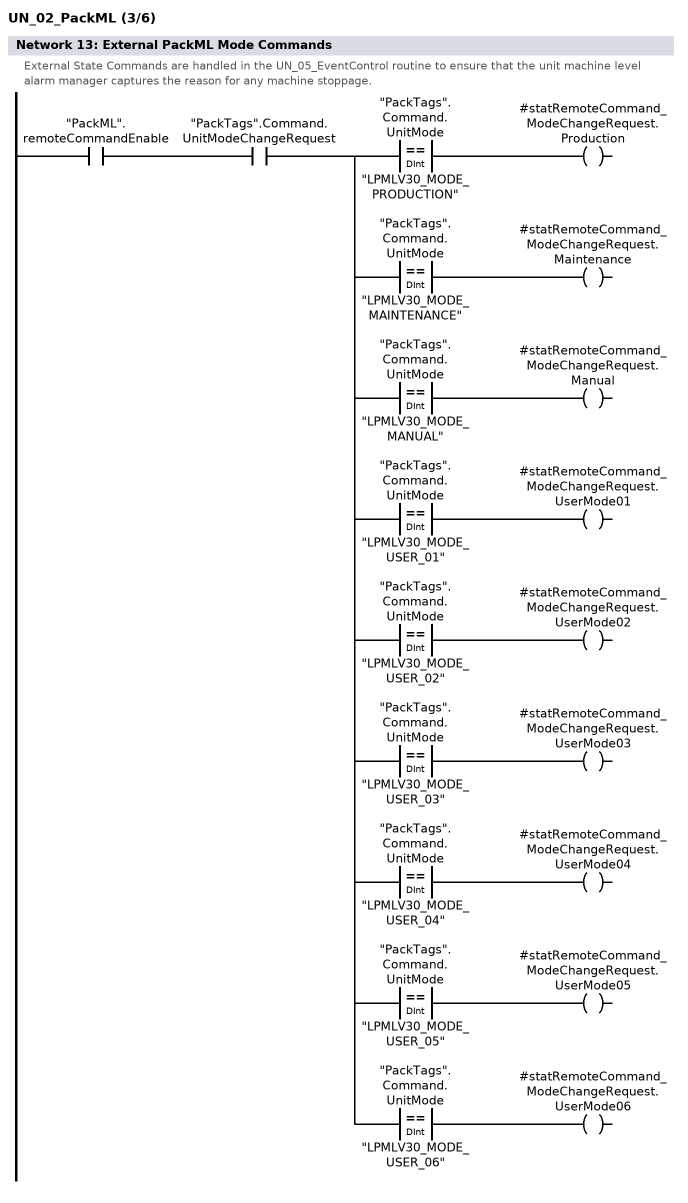
   RUNG wire#powerrail
      Contact( "PackML".remoteCommandEnable )
      Contact( "PackTags".Command.UnitModeChangeRequest )
      wire#w1
      { S7_Templates := "SrcType := DInt" } EQ_Contact(in1 := "PackTags".Command.UnitMode, in2 := "LPMLV30_MODE_PRODUCTION")
      Coil( #statRemoteCommand_ModeChangeRequest.Production )
   END_RUNG
   RUNG wire#w1
      { S7_Templates := "SrcType := DInt" } EQ_Contact(in1 := "PackTags".Command.UnitMode, in2 := "LPMLV30_MODE_MAINTENANCE")
      Coil( #statRemoteCommand_ModeChangeRequest.Maintenance )
   END_RUNG
   RUNG wire#w1
      { S7_Templates := "SrcType := DInt" } EQ_Contact(in1 := "PackTags".Command.UnitMode, in2 := "LPMLV30_MODE_MANUAL")
      Coil( #statRemoteCommand_ModeChangeRequest.Manual )
   END_RUNG
   RUNG wire#w1
      { S7_Templates := "SrcType := DInt" } EQ_Contact(in1 := "PackTags".Command.UnitMode, in2 := "LPMLV30_MODE_USER_01")
      Coil( #statRemoteCommand_ModeChangeRequest.UserMode01 )
   END_RUNG
   RUNG wire#w1
      { S7_Templates := "SrcType := DInt" } EQ_Contact(in1 := "PackTags".Command.UnitMode, in2 := "LPMLV30_MODE_USER_02")
      Coil( #statRemoteCommand_ModeChangeRequest.UserMode02 )
   END_RUNG
   RUNG wire#w1
      { S7_Templates := "SrcType := DInt" } EQ_Contact(in1 := "PackTags".Command.UnitMode, in2 := "LPMLV30_MODE_USER_03")
      Coil( #statRemoteCommand_ModeChangeRequest.UserMode03 )
   END_RUNG
   RUNG wire#w1
      { S7_Templates := "SrcType := DInt" } EQ_Contact(in1 := "PackTags".Command.UnitMode, in2 := "LPMLV30_MODE_USER_04")
      Coil( #statRemoteCommand_ModeChangeRequest.UserMode04 )
   END_RUNG
   RUNG wire#w1
      { S7_Templates := "SrcType := DInt" } EQ_Contact(in1 := "PackTags".Command.UnitMode, in2 := "LPMLV30_MODE_USER_05")
      Coil( #statRemoteCommand_ModeChangeRequest.UserMode05 )
   END_RUNG
   RUNG wire#w1
      { S7_Templates := "SrcType := DInt" } EQ_Contact(in1 := "PackTags".Command.UnitMode, in2 := "LPMLV30_MODE_USER_06")
      Coil( #statRemoteCommand_ModeChangeRequest.UserMode06 )
   END_RUNG
   // the same network as SCL:
   #_w1 := "PackML".remoteCommandEnable AND "PackTags".Command.UnitModeChangeRequest;
   #statRemoteCommand_ModeChangeRequest.Production := #_w1 AND ("PackTags".Command.UnitMode = "LPMLV30_MODE_PRODUCTION");
   #statRemoteCommand_ModeChangeRequest.Maintenance := #_w1 AND ("PackTags".Command.UnitMode = "LPMLV30_MODE_MAINTENANCE");
   #statRemoteCommand_ModeChangeRequest.Manual := #_w1 AND ("PackTags".Command.UnitMode = "LPMLV30_MODE_MANUAL");
   #statRemoteCommand_ModeChangeRequest.UserMode01 := #_w1 AND ("PackTags".Command.UnitMode = "LPMLV30_MODE_USER_01");
   #statRemoteCommand_ModeChangeRequest.UserMode02 := #_w1 AND ("PackTags".Command.UnitMode = "LPMLV30_MODE_USER_02");
   #statRemoteCommand_ModeChangeRequest.UserMode03 := #_w1 AND ("PackTags".Command.UnitMode = "LPMLV30_MODE_USER_03");
   #statRemoteCommand_ModeChangeRequest.UserMode04 := #_w1 AND ("PackTags".Command.UnitMode = "LPMLV30_MODE_USER_04");
   #statRemoteCommand_ModeChangeRequest.UserMode05 := #_w1 AND ("PackTags".Command.UnitMode = "LPMLV30_MODE_USER_05");
   #statRemoteCommand_ModeChangeRequest.UserMode06 := #_w1 AND ("PackTags".Command.UnitMode = "LPMLV30_MODE_USER_06");
END_REGION

REGION Network 14: Call thePackML Mode Manager & State Model FB
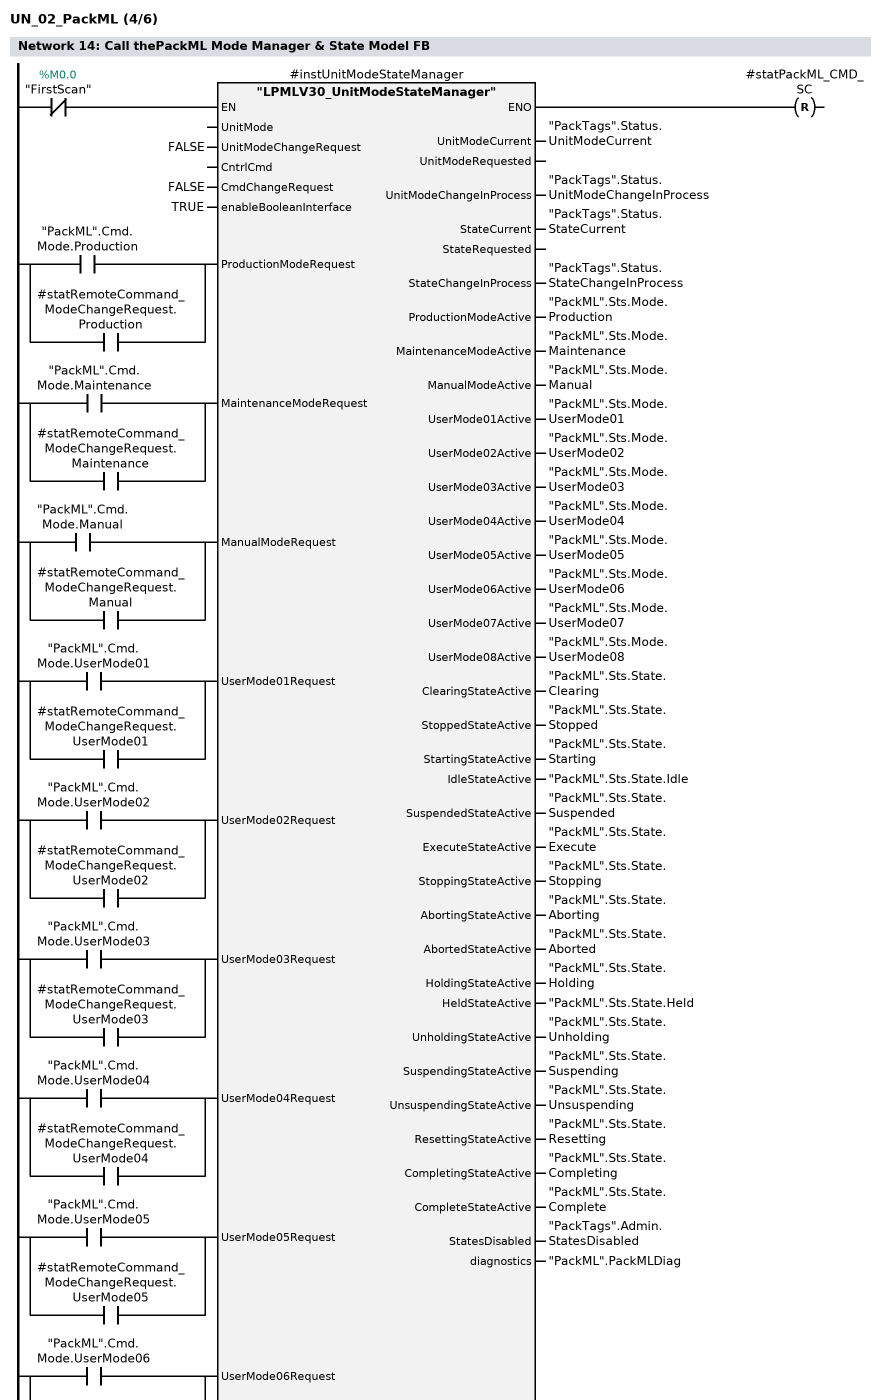
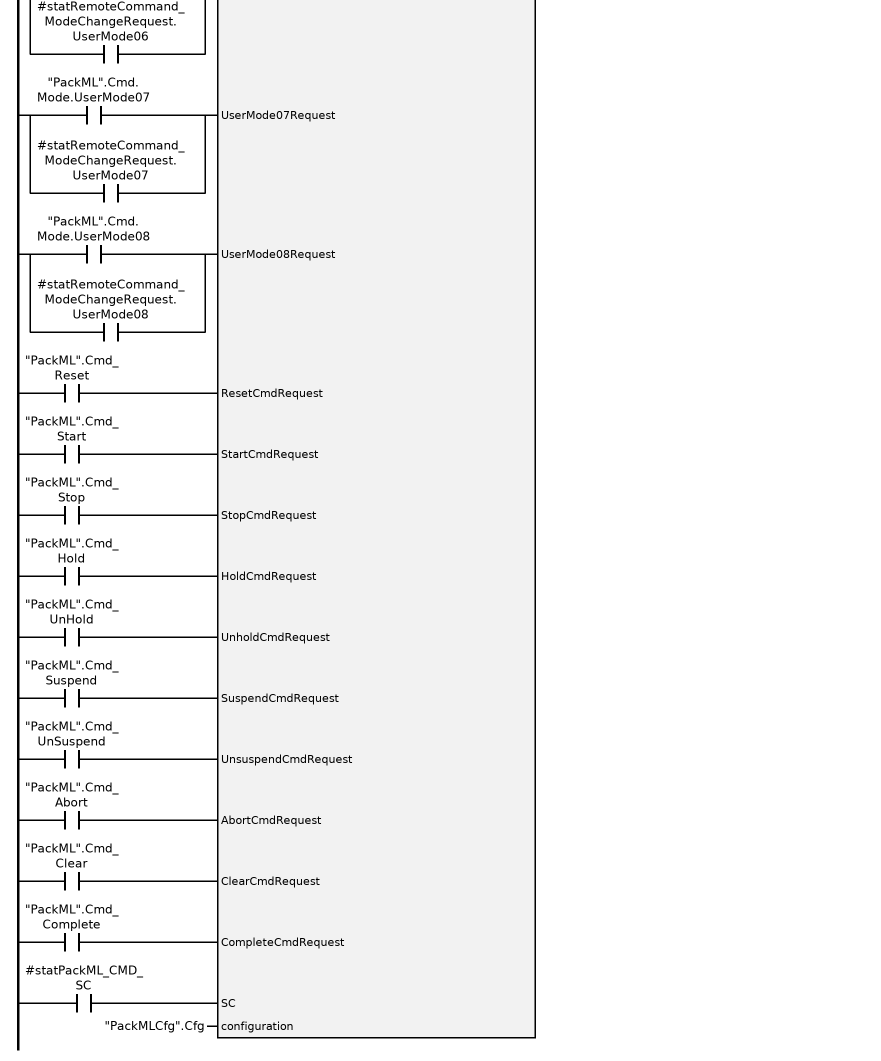
   RUNG wire#powerrail
      I_Contact( "FirstScan" )
      #instUnitModeStateManager(ProductionModeRequest := wire#w1, MaintenanceModeRequest := wire#w2, ManualModeRequest := wire#w3, UserMode01Request := wire#w4, UserMode02Request := wire#w5, UserMode03Request := wire#w6, UserMode04Request := wire#w7, UserMode05Request := wire#w8, UserMode06Request := wire#w9, UserMode07Request := wire#w10, UserMode08Request := wire#w11, ResetCmdRequest := wire#w12, StartCmdRequest := wire#w13, StopCmdRequest := wire#w14, HoldCmdRequest := wire#w15, UnholdCmdRequest := wire#w16, SuspendCmdRequest := wire#w17, UnsuspendCmdRequest := wire#w18, AbortCmdRequest := wire#w19, ClearCmdRequest := wire#w20, CompleteCmdRequest := wire#w21, SC := wire#w22, UnitMode :=, UnitModeChangeRequest := FALSE, CntrlCmd :=, CmdChangeRequest := FALSE, enableBooleanInterface := TRUE, configuration := "PackMLCfg".Cfg, UnitModeCurrent => "PackTags".Status.UnitModeCurrent, UnitModeRequested =>, UnitModeChangeInProcess => "PackTags".Status.UnitModeChangeInProcess, StateCurrent => "PackTags".Status.StateCurrent, StateRequested =>, StateChangeInProcess => "PackTags".Status.StateChangeInProcess, ProductionModeActive => "PackML".Sts.Mode.Production, MaintenanceModeActive => "PackML".Sts.Mode.Maintenance, ManualModeActive => "PackML".Sts.Mode.Manual, UserMode01Active => "PackML".Sts.Mode.UserMode01, UserMode02Active => "PackML".Sts.Mode.UserMode02, UserMode03Active => "PackML".Sts.Mode.UserMode03, UserMode04Active => "PackML".Sts.Mode.UserMode04, UserMode05Active => "PackML".Sts.Mode.UserMode05, UserMode06Active => "PackML".Sts.Mode.UserMode06, UserMode07Active => "PackML".Sts.Mode.UserMode07, UserMode08Active => "PackML".Sts.Mode.UserMode08, ClearingStateActive => "PackML".Sts.State.Clearing, StoppedStateActive => "PackML".Sts.State.Stopped, StartingStateActive => "PackML".Sts.State.Starting, IdleStateActive => "PackML".Sts.State.Idle, SuspendedStateActive => "PackML".Sts.State.Suspended, ExecuteStateActive => "PackML".Sts.State.Execute, StoppingStateActive => "PackML".Sts.State.Stopping, AbortingStateActive => "PackML".Sts.State.Aborting, AbortedStateActive => "PackML".Sts.State.Aborted, HoldingStateActive => "PackML".Sts.State.Holding, HeldStateActive => "PackML".Sts.State.Held, UnholdingStateActive => "PackML".Sts.State.Unholding, SuspendingStateActive => "PackML".Sts.State.Suspending, UnsuspendingStateActive => "PackML".Sts.State.Unsuspending, ResettingStateActive => "PackML".Sts.State.Resetting, CompletingStateActive => "PackML".Sts.State.Completing, CompleteStateActive => "PackML".Sts.State.Complete, StatesDisabled => "PackTags".Admin.StatesDisabled, diagnostics => "PackML".PackMLDiag)
      R_Coil( #statPackML_CMD_SC )
   END_RUNG
   RUNG wire#powerrail
      Contact( "PackML".Cmd.Mode.Production )
   END_RUNG wire#w1
   RUNG wire#powerrail
      Contact( #statRemoteCommand_ModeChangeRequest.Production )
   END_RUNG wire#w1
   RUNG wire#powerrail
      Contact( "PackML".Cmd.Mode.Maintenance )
   END_RUNG wire#w2
   RUNG wire#powerrail
      Contact( #statRemoteCommand_ModeChangeRequest.Maintenance )
   END_RUNG wire#w2
   RUNG wire#powerrail
      Contact( "PackML".Cmd.Mode.Manual )
   END_RUNG wire#w3
   RUNG wire#powerrail
      Contact( #statRemoteCommand_ModeChangeRequest.Manual )
   END_RUNG wire#w3
   RUNG wire#powerrail
      Contact( "PackML".Cmd.Mode.UserMode01 )
   END_RUNG wire#w4
   RUNG wire#powerrail
      Contact( #statRemoteCommand_ModeChangeRequest.UserMode01 )
   END_RUNG wire#w4
   RUNG wire#powerrail
      Contact( "PackML".Cmd.Mode.UserMode02 )
   END_RUNG wire#w5
   RUNG wire#powerrail
      Contact( #statRemoteCommand_ModeChangeRequest.UserMode02 )
   END_RUNG wire#w5
   RUNG wire#powerrail
      Contact( "PackML".Cmd.Mode.UserMode03 )
   END_RUNG wire#w6
   RUNG wire#powerrail
      Contact( #statRemoteCommand_ModeChangeRequest.UserMode03 )
   END_RUNG wire#w6
   RUNG wire#powerrail
      Contact( "PackML".Cmd.Mode.UserMode04 )
   END_RUNG wire#w7
   RUNG wire#powerrail
      Contact( #statRemoteCommand_ModeChangeRequest.UserMode04 )
   END_RUNG wire#w7
   RUNG wire#powerrail
      Contact( "PackML".Cmd.Mode.UserMode05 )
   END_RUNG wire#w8
   RUNG wire#powerrail
      Contact( #statRemoteCommand_ModeChangeRequest.UserMode05 )
   END_RUNG wire#w8
   RUNG wire#powerrail
      Contact( "PackML".Cmd.Mode.UserMode06 )
   END_RUNG wire#w9
   RUNG wire#powerrail
      Contact( #statRemoteCommand_ModeChangeRequest.UserMode06 )
   END_RUNG wire#w9
   RUNG wire#powerrail
      Contact( "PackML".Cmd.Mode.UserMode07 )
   END_RUNG wire#w10
   RUNG wire#powerrail
      Contact( #statRemoteCommand_ModeChangeRequest.UserMode07 )
   END_RUNG wire#w10
   RUNG wire#powerrail
      Contact( "PackML".Cmd.Mode.UserMode08 )
   END_RUNG wire#w11
   RUNG wire#powerrail
      Contact( #statRemoteCommand_ModeChangeRequest.UserMode08 )
   END_RUNG wire#w11
   RUNG wire#powerrail
      Contact( "PackML".Cmd_Reset )
   END_RUNG wire#w12
   RUNG wire#powerrail
      Contact( "PackML".Cmd_Start )
   END_RUNG wire#w13
   RUNG wire#powerrail
      Contact( "PackML".Cmd_Stop )
   END_RUNG wire#w14
   RUNG wire#powerrail
      Contact( "PackML".Cmd_Hold )
   END_RUNG wire#w15
   RUNG wire#powerrail
      Contact( "PackML".Cmd_UnHold )
   END_RUNG wire#w16
   RUNG wire#powerrail
      Contact( "PackML".Cmd_Suspend )
   END_RUNG wire#w17
   RUNG wire#powerrail
      Contact( "PackML".Cmd_UnSuspend )
   END_RUNG wire#w18
   RUNG wire#powerrail
      Contact( "PackML".Cmd_Abort )
   END_RUNG wire#w19
   RUNG wire#powerrail
      Contact( "PackML".Cmd_Clear )
   END_RUNG wire#w20
   RUNG wire#powerrail
      Contact( "PackML".Cmd_Complete )
   END_RUNG wire#w21
   RUNG wire#powerrail
      Contact( #statPackML_CMD_SC )
   END_RUNG wire#w22
   // the same network as SCL:
   #instUnitModeStateManager(EN := NOT "FirstScan",   // "LPMLV30_UnitModeStateManager"
                           UnitModeChangeRequest := FALSE,
                           CmdChangeRequest := FALSE,
                           enableBooleanInterface := TRUE,
                           ProductionModeRequest := "PackML".Cmd.Mode.Production OR #statRemoteCommand_ModeChangeRequest.Production,
                           MaintenanceModeRequest := "PackML".Cmd.Mode.Maintenance OR #statRemoteCommand_ModeChangeRequest.Maintenance,
                           ManualModeRequest := "PackML".Cmd.Mode.Manual OR #statRemoteCommand_ModeChangeRequest.Manual,
                           UserMode01Request := "PackML".Cmd.Mode.UserMode01 OR #statRemoteCommand_ModeChangeRequest.UserMode01,
                           UserMode02Request := "PackML".Cmd.Mode.UserMode02 OR #statRemoteCommand_ModeChangeRequest.UserMode02,
                           UserMode03Request := "PackML".Cmd.Mode.UserMode03 OR #statRemoteCommand_ModeChangeRequest.UserMode03,
                           UserMode04Request := "PackML".Cmd.Mode.UserMode04 OR #statRemoteCommand_ModeChangeRequest.UserMode04,
                           UserMode05Request := "PackML".Cmd.Mode.UserMode05 OR #statRemoteCommand_ModeChangeRequest.UserMode05,
                           UserMode06Request := "PackML".Cmd.Mode.UserMode06 OR #statRemoteCommand_ModeChangeRequest.UserMode06,
                           UserMode07Request := "PackML".Cmd.Mode.UserMode07 OR #statRemoteCommand_ModeChangeRequest.UserMode07,
                           UserMode08Request := "PackML".Cmd.Mode.UserMode08 OR #statRemoteCommand_ModeChangeRequest.UserMode08,
                           ResetCmdRequest := "PackML".Cmd_Reset,
                           StartCmdRequest := "PackML".Cmd_Start,
                           StopCmdRequest := "PackML".Cmd_Stop,
                           HoldCmdRequest := "PackML".Cmd_Hold,
                           UnholdCmdRequest := "PackML".Cmd_UnHold,
                           SuspendCmdRequest := "PackML".Cmd_Suspend,
                           UnsuspendCmdRequest := "PackML".Cmd_UnSuspend,
                           AbortCmdRequest := "PackML".Cmd_Abort,
                           ClearCmdRequest := "PackML".Cmd_Clear,
                           CompleteCmdRequest := "PackML".Cmd_Complete,
                           SC := #statPackML_CMD_SC,
                           configuration := "PackMLCfg".Cfg,
                           UnitModeCurrent => "PackTags".Status.UnitModeCurrent,
                           UnitModeChangeInProcess => "PackTags".Status.UnitModeChangeInProcess,
                           StateCurrent => "PackTags".Status.StateCurrent,
                           StateChangeInProcess => "PackTags".Status.StateChangeInProcess,
                           ProductionModeActive => "PackML".Sts.Mode.Production,
                           MaintenanceModeActive => "PackML".Sts.Mode.Maintenance,
                           ManualModeActive => "PackML".Sts.Mode.Manual,
                           UserMode01Active => "PackML".Sts.Mode.UserMode01,
                           UserMode02Active => "PackML".Sts.Mode.UserMode02,
                           UserMode03Active => "PackML".Sts.Mode.UserMode03,
                           UserMode04Active => "PackML".Sts.Mode.UserMode04,
                           UserMode05Active => "PackML".Sts.Mode.UserMode05,
                           UserMode06Active => "PackML".Sts.Mode.UserMode06,
                           UserMode07Active => "PackML".Sts.Mode.UserMode07,
                           UserMode08Active => "PackML".Sts.Mode.UserMode08,
                           ClearingStateActive => "PackML".Sts.State.Clearing,
                           StoppedStateActive => "PackML".Sts.State.Stopped,
                           StartingStateActive => "PackML".Sts.State.Starting,
                           IdleStateActive => "PackML".Sts.State.Idle,
                           SuspendedStateActive => "PackML".Sts.State.Suspended,
                           ExecuteStateActive => "PackML".Sts.State.Execute,
                           StoppingStateActive => "PackML".Sts.State.Stopping,
                           AbortingStateActive => "PackML".Sts.State.Aborting,
                           AbortedStateActive => "PackML".Sts.State.Aborted,
                           HoldingStateActive => "PackML".Sts.State.Holding,
                           HeldStateActive => "PackML".Sts.State.Held,
                           UnholdingStateActive => "PackML".Sts.State.Unholding,
                           SuspendingStateActive => "PackML".Sts.State.Suspending,
                           UnsuspendingStateActive => "PackML".Sts.State.Unsuspending,
                           ResettingStateActive => "PackML".Sts.State.Resetting,
                           CompletingStateActive => "PackML".Sts.State.Completing,
                           CompleteStateActive => "PackML".Sts.State.Complete,
                           StatesDisabled => "PackTags".Admin.StatesDisabled,
                           diagnostics => "PackML".PackMLDiag,
                           ENO => #_w1);
   IF #_w1 THEN #statPackML_CMD_SC := FALSE; END_IF;
END_REGION

REGION Network 15: "Times" used to format PackML.Admin times and for the HMI display
   // PackML State and Mode Times for HMI
   // 
   // The times spent in each mode and state are calculated in the PackML FB.  This 
   // FB is used to move the modes and states time arrays (current and cumulative 
   // times) into a single array - that is based upon the curent mode - for both 
   // current and cumlative state times.   This single arry is used by the HMI
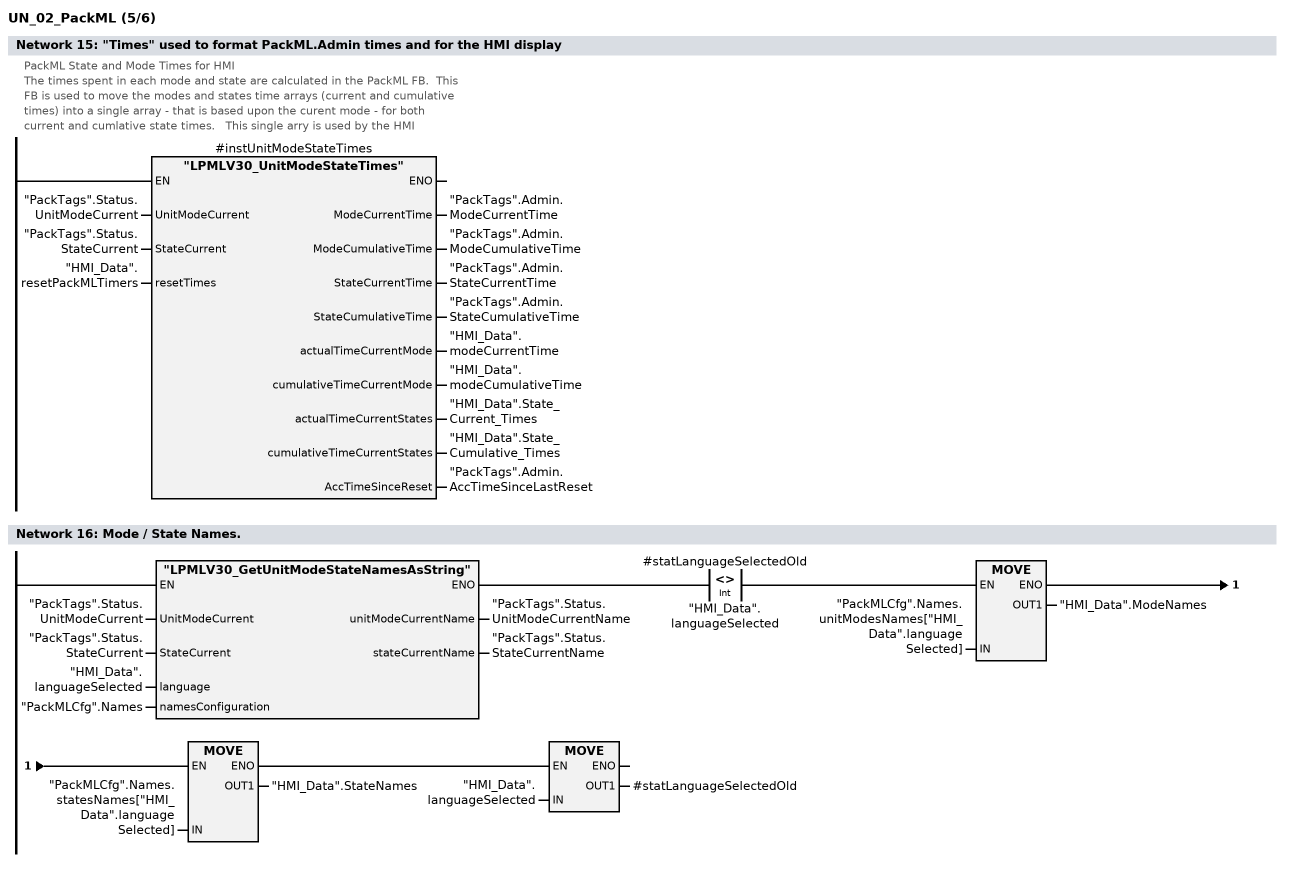
   RUNG wire#powerrail
      #instUnitModeStateTimes(UnitModeCurrent := "PackTags".Status.UnitModeCurrent, StateCurrent := "PackTags".Status.StateCurrent, resetTimes := "HMI_Data".resetPackMLTimers, ModeCurrentTime => "PackTags".Admin.ModeCurrentTime, ModeCumulativeTime => "PackTags".Admin.ModeCumulativeTime, StateCurrentTime => "PackTags".Admin.StateCurrentTime, StateCumulativeTime => "PackTags".Admin.StateCumulativeTime, actualTimeCurrentMode => "HMI_Data".modeCurrentTime, cumulativeTimeCurrentMode => "HMI_Data".modeCumulativeTime, actualTimeCurrentStates => "HMI_Data".State_Current_Times, cumulativeTimeCurrentStates => "HMI_Data".State_Cumulative_Times, AccTimeSinceReset => "PackTags".Admin.AccTimeSinceLastReset)
   END_RUNG
   // the same network as SCL:
   #instUnitModeStateTimes(UnitModeCurrent := "PackTags".Status.UnitModeCurrent,   // "LPMLV30_UnitModeStateTimes"
                           StateCurrent := "PackTags".Status.StateCurrent,
                           resetTimes := "HMI_Data".resetPackMLTimers,
                           ModeCurrentTime => "PackTags".Admin.ModeCurrentTime,
                           ModeCumulativeTime => "PackTags".Admin.ModeCumulativeTime,
                           StateCurrentTime => "PackTags".Admin.StateCurrentTime,
                           StateCumulativeTime => "PackTags".Admin.StateCumulativeTime,
                           actualTimeCurrentMode => "HMI_Data".modeCurrentTime,
                           cumulativeTimeCurrentMode => "HMI_Data".modeCumulativeTime,
                           actualTimeCurrentStates => "HMI_Data".State_Current_Times,
                           cumulativeTimeCurrentStates => "HMI_Data".State_Cumulative_Times,
                           AccTimeSinceReset => "PackTags".Admin.AccTimeSinceLastReset);
END_REGION

REGION Network 16: Mode / State Names.
   RUNG wire#powerrail
      "LPMLV30_GetUnitModeStateNamesAsString"(UnitModeCurrent := "PackTags".Status.UnitModeCurrent, StateCurrent := "PackTags".Status.StateCurrent, language := "HMI_Data".languageSelected, namesConfiguration := "PackMLCfg".Names, unitModeCurrentName => "PackTags".Status.UnitModeCurrentName, stateCurrentName => "PackTags".Status.StateCurrentName)
      { S7_Templates := "SrcType := Int" } NE_Contact(in1 := #statLanguageSelectedOld, in2 := "HMI_Data".languageSelected)
      Move(in := "PackMLCfg".Names.unitModesNames["HMI_Data".languageSelected], out1 => "HMI_Data".ModeNames)
      Move(in := "PackMLCfg".Names.statesNames["HMI_Data".languageSelected], out1 => "HMI_Data".StateNames)
      Move(in := "HMI_Data".languageSelected, out1 => #statLanguageSelectedOld)
   END_RUNG
   // the same network as SCL:
   "LPMLV30_GetUnitModeStateNamesAsString"(UnitModeCurrent := "PackTags".Status.UnitModeCurrent,
                           StateCurrent := "PackTags".Status.StateCurrent,
                           language := "HMI_Data".languageSelected,
                           namesConfiguration := "PackMLCfg".Names,
                           unitModeCurrentName => "PackTags".Status.UnitModeCurrentName,
                           stateCurrentName => "PackTags".Status.StateCurrentName,
                           ENO => #_w1);
   IF #_w1 AND (#statLanguageSelectedOld <> "HMI_Data".languageSelected) THEN
       "HMI_Data".ModeNames := "PackMLCfg".Names.unitModesNames["HMI_Data".languageSelected];
       "HMI_Data".StateNames := "PackMLCfg".Names.statesNames["HMI_Data".languageSelected];
       #statLanguageSelectedOld := "HMI_Data".languageSelected;
   END_IF;
END_REGION

REGION Network 17: State Complete Commands
END_REGION

REGION Network 18: Set the State Complete (SC) bit
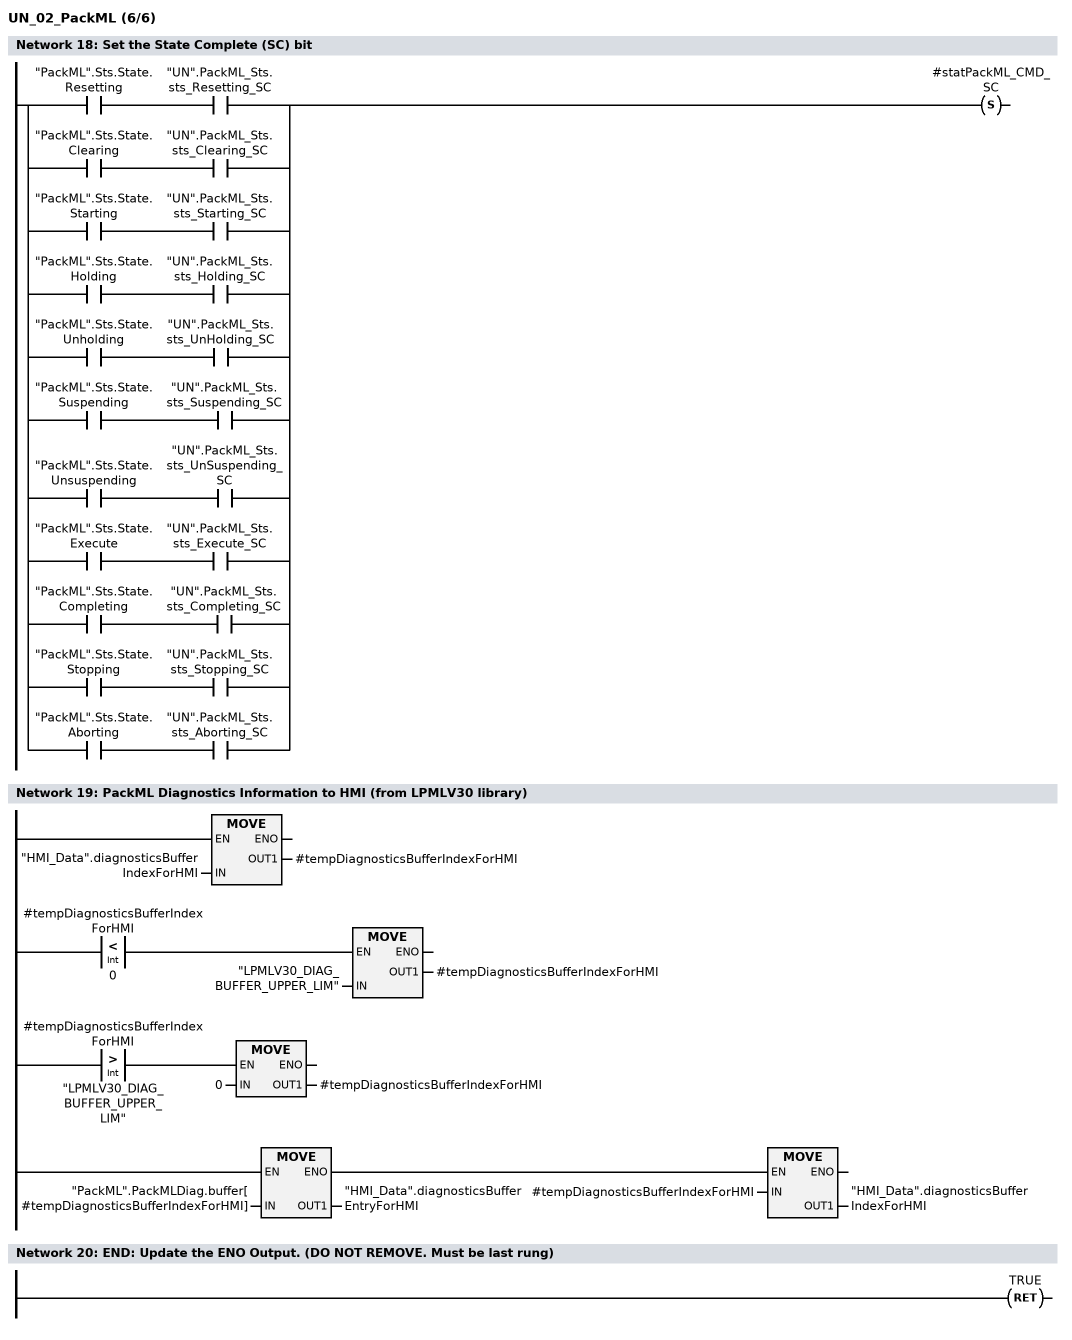
   RUNG wire#powerrail
      Contact( "PackML".Sts.State.Resetting )
      Contact( "UN".PackML_Sts.sts_Resetting_SC )
      wire#w1
      S_Coil( #statPackML_CMD_SC )
   END_RUNG
   RUNG wire#powerrail
      Contact( "PackML".Sts.State.Clearing )
      Contact( "UN".PackML_Sts.sts_Clearing_SC )
   END_RUNG wire#w1
   RUNG wire#powerrail
      Contact( "PackML".Sts.State.Starting )
      Contact( "UN".PackML_Sts.sts_Starting_SC )
   END_RUNG wire#w1
   RUNG wire#powerrail
      Contact( "PackML".Sts.State.Holding )
      Contact( "UN".PackML_Sts.sts_Holding_SC )
   END_RUNG wire#w1
   RUNG wire#powerrail
      Contact( "PackML".Sts.State.Unholding )
      Contact( "UN".PackML_Sts.sts_UnHolding_SC )
   END_RUNG wire#w1
   RUNG wire#powerrail
      Contact( "PackML".Sts.State.Suspending )
      Contact( "UN".PackML_Sts.sts_Suspending_SC )
   END_RUNG wire#w1
   RUNG wire#powerrail
      Contact( "PackML".Sts.State.Unsuspending )
      Contact( "UN".PackML_Sts.sts_UnSuspending_SC )
   END_RUNG wire#w1
   RUNG wire#powerrail
      Contact( "PackML".Sts.State.Execute )
      Contact( "UN".PackML_Sts.sts_Execute_SC )
   END_RUNG wire#w1
   RUNG wire#powerrail
      Contact( "PackML".Sts.State.Completing )
      Contact( "UN".PackML_Sts.sts_Completing_SC )
   END_RUNG wire#w1
   RUNG wire#powerrail
      Contact( "PackML".Sts.State.Stopping )
      Contact( "UN".PackML_Sts.sts_Stopping_SC )
   END_RUNG wire#w1
   RUNG wire#powerrail
      Contact( "PackML".Sts.State.Aborting )
      Contact( "UN".PackML_Sts.sts_Aborting_SC )
   END_RUNG wire#w1
   // the same network as SCL:
   IF ("PackML".Sts.State.Resetting AND "UN".PackML_Sts.sts_Resetting_SC) OR ("PackML".Sts.State.Clearing AND "UN".PackML_Sts.sts_Clearing_SC) OR ("PackML".Sts.State.Starting AND "UN".PackML_Sts.sts_Starting_SC) OR ("PackML".Sts.State.Holding AND "UN".PackML_Sts.sts_Holding_SC) OR ("PackML".Sts.State.Unholding AND "UN".PackML_Sts.sts_UnHolding_SC) OR ("PackML".Sts.State.Suspending AND "UN".PackML_Sts.sts_Suspending_SC) OR ("PackML".Sts.State.Unsuspending AND "UN".PackML_Sts.sts_UnSuspending_SC) OR ("PackML".Sts.State.Execute AND "UN".PackML_Sts.sts_Execute_SC) OR ("PackML".Sts.State.Completing AND "UN".PackML_Sts.sts_Completing_SC) OR ("PackML".Sts.State.Stopping AND "UN".PackML_Sts.sts_Stopping_SC) OR ("PackML".Sts.State.Aborting AND "UN".PackML_Sts.sts_Aborting_SC) THEN
       #statPackML_CMD_SC := TRUE;
   END_IF;
END_REGION

REGION Network 19: PackML Diagnostics Information to HMI (from LPMLV30 library)
   RUNG wire#powerrail
      Move(in := "HMI_Data".diagnosticsBufferIndexForHMI, out1 => #tempDiagnosticsBufferIndexForHMI)
   END_RUNG
   RUNG wire#powerrail
      { S7_Templates := "SrcType := Int" } LT_Contact(in1 := #tempDiagnosticsBufferIndexForHMI, in2 := 0)
      Move(in := "LPMLV30_DIAG_BUFFER_UPPER_LIM", out1 => #tempDiagnosticsBufferIndexForHMI)
   END_RUNG
   RUNG wire#powerrail
      { S7_Templates := "SrcType := Int" } GT_Contact(in1 := #tempDiagnosticsBufferIndexForHMI, in2 := "LPMLV30_DIAG_BUFFER_UPPER_LIM")
      Move(in := 0, out1 => #tempDiagnosticsBufferIndexForHMI)
   END_RUNG
   RUNG wire#powerrail
      Move(in := "PackML".PackMLDiag.buffer[#tempDiagnosticsBufferIndexForHMI], out1 => "HMI_Data".diagnosticsBufferEntryForHMI)
      Move(in := #tempDiagnosticsBufferIndexForHMI, out1 => "HMI_Data".diagnosticsBufferIndexForHMI)
   END_RUNG
   // the same network as SCL:
   #tempDiagnosticsBufferIndexForHMI := "HMI_Data".diagnosticsBufferIndexForHMI;
   IF #tempDiagnosticsBufferIndexForHMI < 0 THEN
       #tempDiagnosticsBufferIndexForHMI := "LPMLV30_DIAG_BUFFER_UPPER_LIM";
   END_IF;
   IF #tempDiagnosticsBufferIndexForHMI > "LPMLV30_DIAG_BUFFER_UPPER_LIM" THEN
       #tempDiagnosticsBufferIndexForHMI := 0;
   END_IF;
   "HMI_Data".diagnosticsBufferEntryForHMI := "PackML".PackMLDiag.buffer[#tempDiagnosticsBufferIndexForHMI];
   "HMI_Data".diagnosticsBufferIndexForHMI := #tempDiagnosticsBufferIndexForHMI;
END_REGION

REGION Network 20: END: Update the ENO Output. (DO NOT REMOVE. Must be last rung)
   RUNG wire#powerrail
      ReturnCoil( TRUE )
   END_RUNG
   // the same network as SCL:
   ENO := TRUE;
   RETURN;
END_REGION
END_FUNCTION_BLOCK

FUNCTION_BLOCK "LPMLV30_UnitModeStateManager"
TITLE = LPMLV30_UnitModeStateManager
{ S7_Optimized_Access := 'TRUE' }
AUTHOR : APC_ERLF
FAMILY : OMAC
//Support: tech.team.motioncontrol@siemens.com 
//Fax: +49 (0) 9131/98-1297
   VAR_INPUT 
      UnitMode : DInt := "LPMLV30_MODE_INVALID";   // Requested unit mode if enableBooleanInterface = FALSE
      UnitModeChangeRequest : Bool := false;   // TRUE: Request unit mode if enableBooleanInterface = FALSE
      CntrlCmd : DInt := "LPMLV30_CMD_UNDEFINED";   // Request control command if enableBooleanInterface = FALSE
      CmdChangeRequest : Bool := false;   // TRUE: Enable change into requested state if enableBooleanInterface = FALSE
      enableBooleanInterface : Bool := false;   // TRUE: Enable boolean interface
      ProductionModeRequest : Bool := false;   // TRUE: Request change to unit mode Production if enableBooleanInterface = TRUE
      MaintenanceModeRequest : Bool := false;   // TRUE: Request change to unit mode Maintenance if enableBooleanInterface = TRUE
      ManualModeRequest : Bool := false;   // TRUE: Request change to unit mode Manual if enableBooleanInterface = TRUE
      UserMode01Request : Bool := false;   // TRUE: Request change to user-defined unit mode 01 if enableBooleanInterface = TRUE
      UserMode02Request : Bool := false;   // TRUE: Request change to user-defined unit mode 02 if enableBooleanInterface = TRUE
      UserMode03Request : Bool := false;   // TRUE: Request change to user-defined unit mode 03 if enableBooleanInterface = TRUE
      UserMode04Request : Bool := false;   // TRUE: Request change to user-defined unit mode 04 if enableBooleanInterface = TRUE
      UserMode05Request : Bool := false;   // TRUE: Request change to user-defined unit mode 05 if enableBooleanInterface = TRUE
      UserMode06Request : Bool := false;   // TRUE: Request change to user-defined unit mode 06 if enableBooleanInterface = TRUE
      UserMode07Request : Bool := false;   // TRUE: Request change to user-defined unit mode 07 if enableBooleanInterface = TRUE
      UserMode08Request : Bool := false;   // TRUE: Request change to user-defined unit mode 08 if enableBooleanInterface = TRUE
      ResetCmdRequest : Bool := false;   // TRUE: Request control command Reset if enableBooleanInterface = TRUE
      StartCmdRequest : Bool := false;   // TRUE: Request control command Start if enableBooleanInterface = TRUE
      StopCmdRequest : Bool := false;   // TRUE: Request control command Stop if enableBooleanInterface = TRUE
      HoldCmdRequest : Bool := false;   // TRUE: Request control command Hold if enableBooleanInterface = TRUE
      UnholdCmdRequest : Bool := false;   // TRUE: Request control command Unhold if enableBooleanInterface = TRUE
      SuspendCmdRequest : Bool := false;   // TRUE: Request control command Suspend if enableBooleanInterface = TRUE
      UnsuspendCmdRequest : Bool := false;   // TRUE: Request control command Unsuspend if enableBooleanInterface = TRUE
      AbortCmdRequest : Bool := false;   // TRUE: Request control command Abort if enableBooleanInterface = TRUE
      ClearCmdRequest : Bool := false;   // TRUE: Request control command Clear if enableBooleanInterface = TRUE
      CompleteCmdRequest : Bool := false;   // TRUE: Request control command Complete if enableBooleanInterface = TRUE
      SC : Bool := false;   // State change from FALSE to TRUE (rising edge) triggers state complete signal
      configuration : "typeLPMLV30_Configuration" := ([12(false), 20(true)], [32(0)]);   // FB configuration
   END_VAR

   VAR_OUTPUT 
      UnitModeCurrent : DInt := "LPMLV30_MODE_MANUAL";   // Current unit mode
      UnitModeRequested : DInt := 0;   // Requested unit mode
      UnitModeChangeInProcess : Bool := false;   // Unit mode change in process
      StateCurrent : DInt := "LPMLV30_STATE_STOPPED";   // Current state
      StateRequested : DInt := 0;   // Requested state
      StateChangeInProcess : Bool := false;   // State change in process
      ProductionModeActive : Bool := false;   // TRUE: Unit mode Production is currently active
      MaintenanceModeActive : Bool := false;   // TRUE: Unit mode Maintenance is currently active
      ManualModeActive : Bool := false;   // TRUE: Unit mode Manual is currently active
      UserMode01Active : Bool := false;   // TRUE: User-defined unit mode 01 is currently active
      UserMode02Active : Bool := false;   // TRUE: User-defined unit mode 02 is currently active
      UserMode03Active : Bool := false;   // TRUE: User-defined unit mode 03 is currently active
      UserMode04Active : Bool := false;   // TRUE: User-defined unit mode 04 is currently active
      UserMode05Active : Bool := false;   // TRUE: User-defined unit mode 05 is currently active
      UserMode06Active : Bool := false;   // TRUE: User-defined unit mode 06 is currently active
      UserMode07Active : Bool := false;   // TRUE: User-defined unit mode 07 is currently active
      UserMode08Active : Bool := false;   // TRUE: User-defined unit mode 08 is currently active
      ClearingStateActive : Bool := false;   // TRUE: State Clearing is currently active
      StoppedStateActive : Bool := false;   // TRUE: State Stopped is currently active
      StartingStateActive : Bool := false;   // TRUE: State Starting is currently active
      IdleStateActive : Bool := false;   // TRUE: State Idle is currently active
      SuspendedStateActive : Bool := false;   // TRUE: State Suspended is currently active
      ExecuteStateActive : Bool := false;   // TRUE: State Execute is currently active
      StoppingStateActive : Bool := false;   // TRUE: State Stopping is currently active
      AbortingStateActive : Bool := false;   // TRUE: State Aborting is currently active
      AbortedStateActive : Bool := false;   // TRUE: State Aborted is currently active
      HoldingStateActive : Bool := false;   // TRUE: State Holding is currently active
      HeldStateActive : Bool := false;   // TRUE: State Held is currently active
      UnholdingStateActive : Bool := false;   // TRUE: State Unholding is currently active
      SuspendingStateActive : Bool := false;   // TRUE: State Suspending is currently active
      UnsuspendingStateActive : Bool := false;   // TRUE: State Unsuspending is currently active
      ResettingStateActive : Bool := false;   // TRUE: State Resetting is currently active
      CompletingStateActive : Bool := false;   // TRUE: State Completing is currently active
      CompleteStateActive : Bool := false;   // TRUE: State Complete is currently active
      StatesDisabled : DInt;   // Disabled states in current unit mode
      diagnostics : "typeLPMLV30_Diagnostics";   // Diagnostics information of FB
   END_VAR

